LIN {X -144.015,Y -42.862,Z -106.683,A -90.000,B 90.000,C 0.000} C_DIS
LIN {X -41.460,Y -42.862,Z -106.683,A -90.000,B 90.000,C 0.000} C_DIS
LIN {X -41.247,Y -42.862,Z -104.786,A -90.000,B 90.000,C 0.000} C_DIS
LIN {X -40.987,Y -42.862,Z -102.895,A -90.000,B 90.000,C 0.000} C_DIS
LIN {X -40.681,Y -42.862,Z -101.010,A -90.000,B 90.000,C 0.000} C_DIS
LIN {X -40.328,Y -42.862,Z -99.134,A -90.000,B 90.000,C 0.000} C_DIS
LIN {X -144.015,Y -42.862,Z -99.134,A -90.000,B 90.000,C 0.000} C_DIS
LIN {X -144.015,Y -42.862,Z -91.586,A -90.000,B 90.000,C 0.000} C_DIS
LIN {X -38.308,Y -42.862,Z -91.586,A -90.000,B 90.000,C 0.000} C_DIS
LIN {X -37.692,Y -42.862,Z -90.026,A -90.000,B 90.000,C 0.000} C_DIS
LIN {X -37.020,Y -42.862,Z -88.489,A -90.000,B 90.000,C 0.000} C_DIS
LIN {X -36.293,Y -42.862,Z -86.977,A -90.000,B 90.000,C 0.000} C_DIS
LIN {X -35.511,Y -42.862,Z -85.492,A -90.000,B 90.000,C 0.000} C_DIS
LIN {X -34.677,Y -42.862,Z -84.037,A -90.000,B 90.000,C 0.000} C_DIS
LIN {X -144.015,Y -42.862,Z -84.037,A -90.000,B 90.000,C 0.000} C_DIS
LIN {X -144.015,Y -42.862,Z -76.488,A -90.000,B 90.000,C 0.000} C_DIS
LIN {X -29.075,Y -42.862,Z -76.488,A -90.000,B 90.000,C 0.000} C_DIS
LIN {X -28.227,Y -42.862,Z -75.567,A -90.000,B 90.000,C 0.000} C_DIS
LIN {X -27.332,Y -42.862,Z -74.692,A -90.000,B 90.000,C 0.000} C_DIS
LIN {X -26.392,Y -42.862,Z -73.865,A -90.000,B 90.000,C 0.000} C_DIS
LIN {X -25.410,Y -42.862,Z -73.089,A -90.000,B 90.000,C 0.000} C_DIS
LIN {X -24.388,Y -42.862,Z -72.366,A -90.000,B 90.000,C 0.000} C_DIS
LIN {X -23.329,Y -42.862,Z -71.698,A -90.000,B 90.000,C 0.000} C_DIS
LIN {X -22.236,Y -42.862,Z -71.087,A -90.000,B 90.000,C 0.000} C_DIS
LIN {X -21.113,Y -42.862,Z -70.535,A -90.000,B 90.000,C 0.000} C_DIS
LIN {X -19.962,Y -42.862,Z -70.043,A -90.000,B 90.000,C 0.000} C_DIS
LIN {X -18.787,Y -42.862,Z -69.612,A -90.000,B 90.000,C 0.000} C_DIS
LIN {X -17.590,Y -42.862,Z -69.244,A -90.000,B 90.000,C 0.000} C_DIS
LIN {X -16.376,Y -42.862,Z -68.939,A -90.000,B 90.000,C 0.000} C_DIS
LIN {X -144.015,Y -42.862,Z -68.939,A -90.000,B 90.000,C 0.000} C_DIS
LIN {X -144.015,Y -42.862,Z -61.390,A -90.000,B 90.000,C 0.000} C_DIS
LIN {X 20.649,Y -42.862,Z -61.390,A -90.000,B 90.000,C 0.000} C_DIS
LIN {X 20.813,Y -42.862,Z -60.536,A -90.000,B 90.000,C 0.000} C_DIS
LIN {X 21.035,Y -42.862,Z -59.695,A -90.000,B 90.000,C 0.000} C_DIS
LIN {X 21.313,Y -42.862,Z -58.871,A -90.000,B 90.000,C 0.000} C_DIS
LIN {X 21.646,Y -42.862,Z -58.068,A -90.000,B 90.000,C 0.000} C_DIS
LIN {X 22.032,Y -42.862,Z -57.289,A -90.000,B 90.000,C 0.000} C_DIS
LIN {X 22.470,Y -42.862,Z -56.537,A -90.000,B 90.000,C 0.000} C_DIS
LIN {X 22.958,Y -42.862,Z -55.817,A -90.000,B 90.000,C 0.000} C_DIS
LIN {X 23.493,Y -42.862,Z -55.132,A -90.000,B 90.000,C 0.000} C_DIS
LIN {X 24.073,Y -42.862,Z -54.484,A -90.000,B 90.000,C 0.000} C_DIS
LIN {X 24.696,Y -42.862,Z -53.877,A -90.000,B 90.000,C 0.000} C_DIS
LIN {X 24.707,Y -42.862,Z -53.842,A -90.000,B 90.000,C 0.000} C_DIS
LIN {X -144.015,Y -42.862,Z -53.842,A -90.000,B 90.000,C 0.000} C_DIS
LIN {X -144.015,Y -42.862,Z -46.293,A -90.000,B 90.000,C 0.000} C_DIS
LIN {X 29.758,Y -42.862,Z -46.293,A -90.000,B 90.000,C 0.000} C_DIS
LIN {X 30.551,Y -42.862,Z -45.689,A -90.000,B 90.000,C 0.000} C_DIS
LIN {X 31.381,Y -42.862,Z -45.138,A -90.000,B 90.000,C 0.000} C_DIS
LIN {X 32.246,Y -42.862,Z -44.643,A -90.000,B 90.000,C 0.000} C_DIS
LIN {X 33.142,Y -42.862,Z -44.206,A -90.000,B 90.000,C 0.000} C_DIS
LIN {X 34.064,Y -42.862,Z -43.828,A -90.000,B 90.000,C 0.000} C_DIS
LIN {X 35.010,Y -42.862,Z -43.513,A -90.000,B 90.000,C 0.000} C_DIS
LIN {X 35.974,Y -42.862,Z -43.260,A -90.000,B 90.000,C 0.000} C_DIS
LIN {X 37.013,Y -42.862,Z -43.088,A -90.000,B 90.000,C 0.000} C_DIS
LIN {X 38.061,Y -42.862,Z -42.978,A -90.000,B 90.000,C 0.000} C_DIS
LIN {X 39.113,Y -42.862,Z -42.931,A -90.000,B 90.000,C 0.000} C_DIS
LIN {X 40.166,Y -42.862,Z -42.946,A -90.000,B 90.000,C 0.000} C_DIS
LIN {X 41.217,Y -42.862,Z -43.023,A -90.000,B 90.000,C 0.000} C_DIS
LIN {X 42.261,Y -42.862,Z -43.163,A -90.000,B 90.000,C 0.000} C_DIS
LIN {X 43.295,Y -42.862,Z -43.364,A -90.000,B 90.000,C 0.000} C_DIS
LIN {X 44.315,Y -42.862,Z -43.626,A -90.000,B 90.000,C 0.000} C_DIS
LIN {X 45.317,Y -42.862,Z -43.948,A -90.000,B 90.000,C 0.000} C_DIS
LIN {X 46.299,Y -42.862,Z -44.329,A -90.000,B 90.000,C 0.000} C_DIS
LIN {X 47.257,Y -42.862,Z -44.768,A -90.000,B 90.000,C 0.000} C_DIS
LIN {X 48.087,Y -42.862,Z -44.686,A -90.000,B 90.000,C 0.000} C_DIS
LIN {X 48.921,Y -42.862,Z -44.656,A -90.000,B 90.000,C 0.000} C_DIS
LIN {X 49.755,Y -42.862,Z -44.677,A -90.000,B 90.000,C 0.000} C_DIS
LIN {X 50.586,Y -42.862,Z -44.750,A -90.000,B 90.000,C 0.000} C_DIS
LIN {X 51.357,Y -42.862,Z -44.828,A -90.000,B 90.000,C 0.000} C_DIS
LIN {X 52.122,Y -42.862,Z -44.958,A -90.000,B 90.000,C 0.000} C_DIS
LIN {X 52.876,Y -42.862,Z -45.137,A -90.000,B 90.000,C 0.000} C_DIS
LIN {X 53.616,Y -42.862,Z -45.367,A -90.000,B 90.000,C 0.000} C_DIS
LIN {X 54.330,Y -42.862,Z -45.538,A -90.000,B 90.000,C 0.000} C_DIS
LIN {X 55.034,Y -42.862,Z -45.750,A -90.000,B 90.000,C 0.000} C_DIS
LIN {X 55.724,Y -42.862,Z -46.002,A -90.000,B 90.000,C 0.000} C_DIS
LIN {X 56.398,Y -42.862,Z -46.293,A -90.000,B 90.000,C 0.000} C_DIS
LIN {X 86.662,Y -42.862,Z -46.293,A -90.000,B 90.000,C 0.000} C_DIS
LIN {X 85.043,Y -42.862,Z -47.710,A -90.000,B 90.000,C 0.000} C_DIS
LIN {X 83.466,Y -42.862,Z -49.175,A -90.000,B 90.000,C 0.000} C_DIS
LIN {X 81.935,Y -42.862,Z -50.686,A -90.000,B 90.000,C 0.000} C_DIS
LIN {X 80.449,Y -42.862,Z -52.242,A -90.000,B 90.000,C 0.000} C_DIS
LIN {X 79.010,Y -42.862,Z -53.842,A -90.000,B 90.000,C 0.000} C_DIS
LIN {X 64.970,Y -42.862,Z -53.842,A -90.000,B 90.000,C 0.000} C_DIS
LIN {X 65.683,Y -42.862,Z -54.842,A -90.000,B 90.000,C 0.000} C_DIS
LIN {X 66.353,Y -42.862,Z -55.871,A -90.000,B 90.000,C 0.000} C_DIS
LIN {X 66.978,Y -42.862,Z -56.928,A -90.000,B 90.000,C 0.000} C_DIS
LIN {X 67.558,Y -42.862,Z -58.010,A -90.000,B 90.000,C 0.000} C_DIS
LIN {X 68.092,Y -42.862,Z -59.116,A -90.000,B 90.000,C 0.000} C_DIS
LIN {X 68.578,Y -42.862,Z -60.243,A -90.000,B 90.000,C 0.000} C_DIS
LIN {X 69.017,Y -42.862,Z -61.390,A -90.000,B 90.000,C 0.000} C_DIS
LIN {X 73.958,Y -42.862,Z -61.390,A -90.000,B 90.000,C 0.000} C_DIS
LIN {X 74.651,Y -42.862,Z -60.082,A -90.000,B 90.000,C 0.000} C_DIS
LIN {X 75.393,Y -42.862,Z -58.802,A -90.000,B 90.000,C 0.000} C_DIS
LIN {X 76.183,Y -42.862,Z -57.550,A -90.000,B 90.000,C 0.000} C_DIS
LIN {X 77.020,Y -42.862,Z -56.330,A -90.000,B 90.000,C 0.000} C_DIS
LIN {X 77.903,Y -42.862,Z -55.142,A -90.000,B 90.000,C 0.000} C_DIS
LIN {X 79.161,Y -42.862,Z -53.670,A -90.000,B 90.000,C 0.000} C_DIS
LIN {X 80.458,Y -42.862,Z -52.232,A -90.000,B 90.000,C 0.000} C_DIS
LIN {X 81.794,Y -42.862,Z -50.830,A -90.000,B 90.000,C 0.000} C_DIS
LIN {X 83.166,Y -42.862,Z -49.464,A -90.000,B 90.000,C 0.000} C_DIS
LIN {X 84.575,Y -42.862,Z -48.136,A -90.000,B 90.000,C 0.000} C_DIS
LIN {X 86.019,Y -42.862,Z -46.846,A -90.000,B 90.000,C 0.000} C_DIS
LIN {X 87.497,Y -42.862,Z -45.595,A -90.000,B 90.000,C 0.000} C_DIS
LIN {X 88.554,Y -42.862,Z -44.745,A -90.000,B 90.000,C 0.000} C_DIS
LIN {X 89.585,Y -42.862,Z -43.865,A -90.000,B 90.000,C 0.000} C_DIS
LIN {X 90.592,Y -42.862,Z -42.956,A -90.000,B 90.000,C 0.000} C_DIS
LIN {X 91.572,Y -42.862,Z -42.019,A -90.000,B 90.000,C 0.000} C_DIS
LIN {X 94.550,Y -42.862,Z -38.744,A -90.000,B 90.000,C 0.000} C_DIS
LIN {X -144.015,Y -42.862,Z -38.744,A -90.000,B 90.000,C 0.000} C_DIS
LIN {X -144.015,Y -42.862,Z -31.195,A -90.000,B 90.000,C 0.000} C_DIS
LIN {X 102.214,Y -42.862,Z -31.195,A -90.000,B 90.000,C 0.000} C_DIS
LIN {X 103.051,Y -42.862,Z -30.607,A -90.000,B 90.000,C 0.000} C_DIS
LIN {X 103.927,Y -42.862,Z -30.078,A -90.000,B 90.000,C 0.000} C_DIS
LIN {X 104.837,Y -42.862,Z -29.611,A -90.000,B 90.000,C 0.000} C_DIS
LIN {X 105.777,Y -42.862,Z -29.208,A -90.000,B 90.000,C 0.000} C_DIS
LIN {X 106.743,Y -42.862,Z -28.871,A -90.000,B 90.000,C 0.000} C_DIS
LIN {X 107.730,Y -42.862,Z -28.602,A -90.000,B 90.000,C 0.000} C_DIS
LIN {X 108.733,Y -42.862,Z -28.401,A -90.000,B 90.000,C 0.000} C_DIS
LIN {X 109.747,Y -42.862,Z -28.270,A -90.000,B 90.000,C 0.000} C_DIS
LIN {X 110.768,Y -42.862,Z -28.209,A -90.000,B 90.000,C 0.000} C_DIS
LIN {X 111.791,Y -42.862,Z -28.219,A -90.000,B 90.000,C 0.000} C_DIS
LIN {X 112.811,Y -42.862,Z -28.301,A -90.000,B 90.000,C 0.000} C_DIS
LIN {X 112.936,Y -42.862,Z -28.324,A -90.000,B 90.000,C 0.000} C_DIS
LIN {X 112.988,Y -42.862,Z -28.327,A -90.000,B 90.000,C 0.000} C_DIS
LIN {X 113.926,Y -42.862,Z -28.470,A -90.000,B 90.000,C 0.000} C_DIS
LIN {X 114.851,Y -42.862,Z -28.677,A -90.000,B 90.000,C 0.000} C_DIS
LIN {X 115.760,Y -42.862,Z -28.948,A -90.000,B 90.000,C 0.000} C_DIS
LIN {X 116.648,Y -42.862,Z -29.280,A -90.000,B 90.000,C 0.000} C_DIS
LIN {X 117.511,Y -42.862,Z -29.673,A -90.000,B 90.000,C 0.000} C_DIS
LIN {X 118.345,Y -42.862,Z -30.125,A -90.000,B 90.000,C 0.000} C_DIS
LIN {X 119.146,Y -42.862,Z -30.633,A -90.000,B 90.000,C 0.000} C_DIS
LIN {X 119.910,Y -42.862,Z -31.195,A -90.000,B 90.000,C 0.000} C_DIS
LIN {X 144.015,Y -42.862,Z -31.195,A -90.000,B 90.000,C 0.000} C_DIS
LIN {X 144.015,Y -42.862,Z -38.744,A -90.000,B 90.000,C 0.000} C_DIS
LIN {X 124.744,Y -42.862,Z -38.744,A -90.000,B 90.000,C 0.000} C_DIS
LIN {X 124.926,Y -42.862,Z -39.587,A -90.000,B 90.000,C 0.000} C_DIS
LIN {X 125.057,Y -42.862,Z -40.439,A -90.000,B 90.000,C 0.000} C_DIS
LIN {X 125.135,Y -42.862,Z -41.298,A -90.000,B 90.000,C 0.000} C_DIS
LIN {X 125.160,Y -42.862,Z -42.159,A -90.000,B 90.000,C 0.000} C_DIS
LIN {X 125.132,Y -42.862,Z -43.021,A -90.000,B 90.000,C 0.000} C_DIS
LIN {X 124.953,Y -42.862,Z -44.119,A -90.000,B 90.000,C 0.000} C_DIS
LIN {X 124.737,Y -42.862,Z -45.210,A -90.000,B 90.000,C 0.000} C_DIS
LIN {X 124.482,Y -42.862,Z -46.293,A -90.000,B 90.000,C 0.000} C_DIS
LIN {X 144.015,Y -42.862,Z -46.293,A -90.000,B 90.000,C 0.000} C_DIS
LIN {X 144.015,Y -42.862,Z -53.842,A -90.000,B 90.000,C 0.000} C_DIS
LIN {X 121.443,Y -42.862,Z -53.842,A -90.000,B 90.000,C 0.000} C_DIS
LIN {X 120.742,Y -42.862,Z -55.297,A -90.000,B 90.000,C 0.000} C_DIS
LIN {X 120.079,Y -42.862,Z -56.770,A -90.000,B 90.000,C 0.000} C_DIS
LIN {X 119.457,Y -42.862,Z -58.260,A -90.000,B 90.000,C 0.000} C_DIS
LIN {X 118.875,Y -42.862,Z -59.766,A -90.000,B 90.000,C 0.000} C_DIS
LIN {X 118.368,Y -42.862,Z -61.390,A -90.000,B 90.000,C 0.000} C_DIS
LIN {X 144.015,Y -42.862,Z -61.390,A -90.000,B 90.000,C 0.000} C_DIS
LIN {X 144.015,Y -42.862,Z -68.939,A -90.000,B 90.000,C 0.000} C_DIS
LIN {X 115.738,Y -42.862,Z -68.939,A -90.000,B 90.000,C 0.000} C_DIS
LIN {X 115.018,Y -42.862,Z -70.802,A -90.000,B 90.000,C 0.000} C_DIS
LIN {X 114.272,Y -42.862,Z -72.655,A -90.000,B 90.000,C 0.000} C_DIS
LIN {X 113.767,Y -42.862,Z -73.946,A -90.000,B 90.000,C 0.000} C_DIS
LIN {X 113.230,Y -42.862,Z -75.224,A -90.000,B 90.000,C 0.000} C_DIS
LIN {X 112.660,Y -42.862,Z -76.488,A -90.000,B 90.000,C 0.000} C_DIS
LIN {X 144.015,Y -42.862,Z -76.488,A -90.000,B 90.000,C 0.000} C_DIS
LIN {X 144.015,Y -42.862,Z -84.037,A -90.000,B 90.000,C 0.000} C_DIS
LIN {X 108.391,Y -42.862,Z -84.037,A -90.000,B 90.000,C 0.000} C_DIS
LIN {X 107.637,Y -42.862,Z -85.126,A -90.000,B 90.000,C 0.000} C_DIS
LIN {X 106.857,Y -42.862,Z -86.197,A -90.000,B 90.000,C 0.000} C_DIS
LIN {X 106.156,Y -42.862,Z -87.168,A -90.000,B 90.000,C 0.000} C_DIS
LIN {X 105.419,Y -42.862,Z -88.112,A -90.000,B 90.000,C 0.000} C_DIS
LIN {X 104.647,Y -42.862,Z -89.027,A -90.000,B 90.000,C 0.000} C_DIS
LIN {X 103.840,Y -42.862,Z -89.911,A -90.000,B 90.000,C 0.000} C_DIS
LIN {X 103.001,Y -42.862,Z -90.765,A -90.000,B 90.000,C 0.000} C_DIS
LIN {X 102.129,Y -42.862,Z -91.586,A -90.000,B 90.000,C 0.000} C_DIS
LIN {X 144.015,Y -42.862,Z -91.586,A -90.000,B 90.000,C 0.000} C_DIS
LIN {X 144.015,Y -42.862,Z -99.134,A -90.000,B 90.000,C 0.000} C_DIS
LIN {X 99.151,Y -42.862,Z -99.134,A -90.000,B 90.000,C 0.000} C_DIS
LIN {X 98.860,Y -42.862,Z -100.099,A -90.000,B 90.000,C 0.000} C_DIS
LIN {X 98.506,Y -42.862,Z -101.043,A -90.000,B 90.000,C 0.000} C_DIS
LIN {X 98.089,Y -42.862,Z -101.961,A -90.000,B 90.000,C 0.000} C_DIS
LIN {X 97.612,Y -42.862,Z -102.849,A -90.000,B 90.000,C 0.000} C_DIS
LIN {X 97.077,Y -42.862,Z -103.703,A -90.000,B 90.000,C 0.000} C_DIS
LIN {X 96.485,Y -42.862,Z -104.519,A -90.000,B 90.000,C 0.000} C_DIS
LIN {X 95.841,Y -42.862,Z -105.294,A -90.000,B 90.000,C 0.000} C_DIS
LIN {X 95.901,Y -42.862,Z -105.988,A -90.000,B 90.000,C 0.000} C_DIS
LIN {X 95.943,Y -42.862,Z -106.683,A -90.000,B 90.000,C 0.000} C_DIS
LIN {X 144.015,Y -42.862,Z -106.683,A -90.000,B 90.000,C 0.000} C_DIS
LIN {X 144.015,Y -42.862,Z -114.232,A -90.000,B 90.000,C 0.000} C_DIS
LIN {X 95.004,Y -42.862,Z -114.232,A -90.000,B 90.000,C 0.000} C_DIS
LIN {X 94.755,Y -42.862,Z -115.216,A -90.000,B 90.000,C 0.000} C_DIS
LIN {X 94.481,Y -42.862,Z -116.194,A -90.000,B 90.000,C 0.000} C_DIS
LIN {X 94.133,Y -42.862,Z -117.126,A -90.000,B 90.000,C 0.000} C_DIS
LIN {X 93.819,Y -42.862,Z -118.070,A -90.000,B 90.000,C 0.000} C_DIS
LIN {X 93.540,Y -42.862,Z -119.025,A -90.000,B 90.000,C 0.000} C_DIS
LIN {X 93.683,Y -42.862,Z -119.949,A -90.000,B 90.000,C 0.000} C_DIS
LIN {X 93.853,Y -42.862,Z -120.868,A -90.000,B 90.000,C 0.000} C_DIS
LIN {X 94.052,Y -42.862,Z -121.781,A -90.000,B 90.000,C 0.000} C_DIS
LIN {X 144.015,Y -42.862,Z -121.781,A -90.000,B 90.000,C 0.000} C_DIS
LIN {X 144.015,Y -42.862,Z -129.329,A -90.000,B 90.000,C 0.000} C_DIS
LIN {X 94.517,Y -42.862,Z -129.329,A -90.000,B 90.000,C 0.000} C_DIS
LIN {X 94.482,Y -42.862,Z -130.307,A -90.000,B 90.000,C 0.000} C_DIS
LIN {X 94.426,Y -42.862,Z -131.284,A -90.000,B 90.000,C 0.000} C_DIS
LIN {X 94.348,Y -42.862,Z -132.259,A -90.000,B 90.000,C 0.000} C_DIS
LIN {X 94.250,Y -42.862,Z -134.569,A -90.000,B 90.000,C 0.000} C_DIS
LIN {X 94.147,Y -42.862,Z -136.878,A -90.000,B 90.000,C 0.000} C_DIS
LIN {X 144.015,Y -42.862,Z -136.878,A -90.000,B 90.000,C 0.000} C_DIS
LIN {X 144.015,Y -42.862,Z -144.427,A -90.000,B 90.000,C 0.000} C_DIS
LIN {X 93.773,Y -42.862,Z -144.427,A -90.000,B 90.000,C 0.000} C_DIS
LIN {X 93.759,Y -42.862,Z -144.687,A -90.000,B 90.000,C 0.000} C_DIS
LIN {X 93.660,Y -42.862,Z -146.513,A -90.000,B 90.000,C 0.000} C_DIS
LIN {X 93.529,Y -42.862,Z -148.337,A -90.000,B 90.000,C 0.000} C_DIS
LIN {X 93.366,Y -42.862,Z -150.158,A -90.000,B 90.000,C 0.000} C_DIS
LIN {X 93.171,Y -42.862,Z -151.976,A -90.000,B 90.000,C 0.000} C_DIS
LIN {X 144.015,Y -42.862,Z -151.976,A -90.000,B 90.000,C 0.000} C_DIS
LIN {X 144.015,Y -42.862,Z -159.525,A -90.000,B 90.000,C 0.000} C_DIS
LIN {X 92.013,Y -42.862,Z -159.525,A -90.000,B 90.000,C 0.000} C_DIS
LIN {X 91.632,Y -42.862,Z -161.424,A -90.000,B 90.000,C 0.000} C_DIS
LIN {X 91.216,Y -42.862,Z -163.315,A -90.000,B 90.000,C 0.000} C_DIS
LIN {X 90.765,Y -42.862,Z -165.198,A -90.000,B 90.000,C 0.000} C_DIS
LIN {X 90.279,Y -42.862,Z -167.073,A -90.000,B 90.000,C 0.000} C_DIS
LIN {X 144.015,Y -42.862,Z -167.073,A -90.000,B 90.000,C 0.000} C_DIS
LIN {X 144.015,Y -42.862,Z -174.622,A -90.000,B 90.000,C 0.000} C_DIS
LIN {X 87.981,Y -42.862,Z -174.622,A -90.000,B 90.000,C 0.000} C_DIS
LIN {X 87.289,Y -42.862,Z -176.815,A -90.000,B 90.000,C 0.000} C_DIS
LIN {X 86.606,Y -42.862,Z -179.011,A -90.000,B 90.000,C 0.000} C_DIS
LIN {X 85.836,Y -42.862,Z -182.171,A -90.000,B 90.000,C 0.000} C_DIS
LIN {X 144.015,Y -42.862,Z -182.171,A -90.000,B 90.000,C 0.000} C_DIS
LIN {X 144.015,Y -42.862,Z -189.720,A -90.000,B 90.000,C 0.000} C_DIS
LIN {X 83.918,Y -42.862,Z -189.720,A -90.000,B 90.000,C 0.000} C_DIS
LIN {X 83.235,Y -42.862,Z -192.307,A -90.000,B 90.000,C 0.000} C_DIS
LIN {X 82.539,Y -42.862,Z -194.890,A -90.000,B 90.000,C 0.000} C_DIS
LIN {X 82.150,Y -42.862,Z -196.080,A -90.000,B 90.000,C 0.000} C_DIS
LIN {X 81.756,Y -42.862,Z -197.269,A -90.000,B 90.000,C 0.000} C_DIS
LIN {X 144.015,Y -42.862,Z -197.269,A -90.000,B 90.000,C 0.000} C_DIS
LIN {X 144.015,Y -42.862,Z -204.817,A -90.000,B 90.000,C 0.000} C_DIS
LIN {X 79.114,Y -42.862,Z -204.817,A -90.000,B 90.000,C 0.000} C_DIS
LIN {X 78.176,Y -42.862,Z -207.342,A -90.000,B 90.000,C 0.000} C_DIS
LIN {X 77.215,Y -42.862,Z -209.859,A -90.000,B 90.000,C 0.000} C_DIS
LIN {X 76.229,Y -42.862,Z -212.366,A -90.000,B 90.000,C 0.000} C_DIS
LIN {X 144.015,Y -42.862,Z -212.366,A -90.000,B 90.000,C 0.000} C_DIS
LIN {X 144.015,Y -42.862,Z -219.915,A -90.000,B 90.000,C 0.000} C_DIS
LIN {X 73.092,Y -42.862,Z -219.915,A -90.000,B 90.000,C 0.000} C_DIS
LIN {X 71.984,Y -42.862,Z -222.442,A -90.000,B 90.000,C 0.000} C_DIS
LIN {X 70.851,Y -42.862,Z -224.959,A -90.000,B 90.000,C 0.000} C_DIS
LIN {X 69.694,Y -42.862,Z -227.464,A -90.000,B 90.000,C 0.000} C_DIS
LIN {X 144.015,Y -42.862,Z -227.464,A -90.000,B 90.000,C 0.000} C_DIS
LIN {X 144.015,Y -42.862,Z -235.012,A -90.000,B 90.000,C 0.000} C_DIS
LIN {X 66.063,Y -42.862,Z -235.012,A -90.000,B 90.000,C 0.000} C_DIS
LIN {X 65.077,Y -42.862,Z -236.924,A -90.000,B 90.000,C 0.000} C_DIS
LIN {X 64.061,Y -42.862,Z -238.820,A -90.000,B 90.000,C 0.000} C_DIS
LIN {X 63.015,Y -42.862,Z -240.699,A -90.000,B 90.000,C 0.000} C_DIS
LIN {X 61.939,Y -42.862,Z -242.561,A -90.000,B 90.000,C 0.000} C_DIS
LIN {X 144.015,Y -42.862,Z -242.561,A -90.000,B 90.000,C 0.000} C_DIS
LIN {X 144.015,Y -42.862,Z -23.646,A -90.000,B 90.000,C 0.000} C_DIS
LIN {X -144.015,Y -42.862,Z -23.646,A -90.000,B 90.000,C 0.000} C_DIS
LIN {X -144.015,Y -42.862,Z -16.098,A -90.000,B 90.000,C 0.000} C_DIS
LIN {X 144.015,Y -42.862,Z -16.098,A -90.000,B 90.000,C 0.000} C_DIS
LIN {X 144.015,Y -42.862,Z -8.549,A -90.000,B 90.000,C 0.000} C_DIS
LIN {X -144.015,Y -42.862,Z -8.549,A -90.000,B 90.000,C 0.000} C_DIS
LIN {X -144.015,Y -42.862,Z -1.000,A -90.000,B 90.000,C 0.000} C_DIS
LIN {X 144.015,Y -42.862,Z -1.000,A -90.000,B 90.000,C 0.000} C_DIS
LIN {X 55.699,Y -42.862,Z -45.992,A -90.000,B 90.000,C 0.000} C_DIS
LIN {X 55.017,Y -42.862,Z -45.744,A -90.000,B 90.000,C 0.000} C_DIS
LIN {X 54.322,Y -42.862,Z -45.536,A -90.000,B 90.000,C 0.000} C_DIS
LIN {X 53.616,Y -42.862,Z -45.367,A -90.000,B 90.000,C 0.000} C_DIS
LIN {X 52.876,Y -42.862,Z -45.138,A -90.000,B 90.000,C 0.000} C_DIS
LIN {X 52.121,Y -42.862,Z -44.958,A -90.000,B 90.000,C 0.000} C_DIS
LIN {X 51.357,Y -42.862,Z -44.829,A -90.000,B 90.000,C 0.000} C_DIS
LIN {X 50.586,Y -42.862,Z -44.750,A -90.000,B 90.000,C 0.000} C_DIS
LIN {X 49.755,Y -42.862,Z -44.677,A -90.000,B 90.000,C 0.000} C_DIS
LIN {X 48.921,Y -42.862,Z -44.656,A -90.000,B 90.000,C 0.000} C_DIS
LIN {X 48.087,Y -42.862,Z -44.687,A -90.000,B 90.000,C 0.000} C_DIS
LIN {X 47.257,Y -42.862,Z -44.768,A -90.000,B 90.000,C 0.000} C_DIS
LIN {X 46.299,Y -42.862,Z -44.329,A -90.000,B 90.000,C 0.000} C_DIS
LIN {X 45.317,Y -42.862,Z -43.948,A -90.000,B 90.000,C 0.000} C_DIS
LIN {X 44.315,Y -42.862,Z -43.626,A -90.000,B 90.000,C 0.000} C_DIS
LIN {X 43.295,Y -42.862,Z -43.364,A -90.000,B 90.000,C 0.000} C_DIS
LIN {X 42.261,Y -42.862,Z -43.163,A -90.000,B 90.000,C 0.000} C_DIS
LIN {X 41.217,Y -42.862,Z -43.023,A -90.000,B 90.000,C 0.000} C_DIS
LIN {X 40.166,Y -42.862,Z -42.946,A -90.000,B 90.000,C 0.000} C_DIS
LIN {X 39.113,Y -42.862,Z -42.931,A -90.000,B 90.000,C 0.000} C_DIS
LIN {X 38.061,Y -42.862,Z -42.978,A -90.000,B 90.000,C 0.000} C_DIS
LIN {X 37.013,Y -42.862,Z -43.088,A -90.000,B 90.000,C 0.000} C_DIS
LIN {X 35.974,Y -42.862,Z -43.260,A -90.000,B 90.000,C 0.000} C_DIS
LIN {X 34.989,Y -42.862,Z -43.519,A -90.000,B 90.000,C 0.000} C_DIS
LIN {X 34.023,Y -42.862,Z -43.844,A -90.000,B 90.000,C 0.000} C_DIS
LIN {X 33.082,Y -42.862,Z -44.233,A -90.000,B 90.000,C 0.000} C_DIS
LIN {X 32.168,Y -42.862,Z -44.684,A -90.000,B 90.000,C 0.000} C_DIS
LIN {X 31.287,Y -42.862,Z -45.196,A -90.000,B 90.000,C 0.000} C_DIS
LIN {X 30.443,Y -42.862,Z -45.766,A -90.000,B 90.000,C 0.000} C_DIS
LIN {X 29.639,Y -42.862,Z -46.391,A -90.000,B 90.000,C 0.000} C_DIS
LIN {X 28.879,Y -42.862,Z -47.069,A -90.000,B 90.000,C 0.000} C_DIS
LIN {X 28.166,Y -42.862,Z -47.797,A -90.000,B 90.000,C 0.000} C_DIS
LIN {X 27.503,Y -42.862,Z -48.571,A -90.000,B 90.000,C 0.000} C_DIS
LIN {X 26.894,Y -42.862,Z -49.388,A -90.000,B 90.000,C 0.000} C_DIS
LIN {X 26.342,Y -42.862,Z -50.244,A -90.000,B 90.000,C 0.000} C_DIS
LIN {X 25.848,Y -42.862,Z -51.135,A -90.000,B 90.000,C 0.000} C_DIS
LIN {X 25.415,Y -42.862,Z -52.057,A -90.000,B 90.000,C 0.000} C_DIS
LIN {X 25.138,Y -42.862,Z -52.649,A -90.000,B 90.000,C 0.000} C_DIS
LIN {X 24.898,Y -42.862,Z -53.256,A -90.000,B 90.000,C 0.000} C_DIS
LIN {X 24.696,Y -42.862,Z -53.877,A -90.000,B 90.000,C 0.000} C_DIS
LIN {X 24.058,Y -42.862,Z -54.500,A -90.000,B 90.000,C 0.000} C_DIS
LIN {X 23.464,Y -42.862,Z -55.167,A -90.000,B 90.000,C 0.000} C_DIS
LIN {X 22.918,Y -42.862,Z -55.872,A -90.000,B 90.000,C 0.000} C_DIS
LIN {X 22.422,Y -42.862,Z -56.614,A -90.000,B 90.000,C 0.000} C_DIS
LIN {X 21.979,Y -42.862,Z -57.388,A -90.000,B 90.000,C 0.000} C_DIS
LIN {X 21.590,Y -42.862,Z -58.191,A -90.000,B 90.000,C 0.000} C_DIS
LIN {X 21.258,Y -42.862,Z -59.020,A -90.000,B 90.000,C 0.000} C_DIS
LIN {X 20.984,Y -42.862,Z -59.869,A -90.000,B 90.000,C 0.000} C_DIS
LIN {X 20.770,Y -42.862,Z -60.735,A -90.000,B 90.000,C 0.000} C_DIS
LIN {X 20.616,Y -42.862,Z -61.614,A -90.000,B 90.000,C 0.000} C_DIS
LIN {X 20.523,Y -42.862,Z -62.501,A -90.000,B 90.000,C 0.000} C_DIS
LIN {X 19.836,Y -42.862,Z -62.571,A -90.000,B 90.000,C 0.000} C_DIS
LIN {X 19.155,Y -42.862,Z -62.686,A -90.000,B 90.000,C 0.000} C_DIS
LIN {X 18.482,Y -42.862,Z -62.843,A -90.000,B 90.000,C 0.000} C_DIS
LIN {X 18.425,Y -42.862,Z -62.863,A -90.000,B 90.000,C 0.000} C_DIS
LIN {X 17.595,Y -42.862,Z -63.039,A -90.000,B 90.000,C 0.000} C_DIS
LIN {X 16.783,Y -42.862,Z -63.284,A -90.000,B 90.000,C 0.000} C_DIS
LIN {X 15.994,Y -42.862,Z -63.595,A -90.000,B 90.000,C 0.000} C_DIS
LIN {X 15.234,Y -42.862,Z -63.970,A -90.000,B 90.000,C 0.000} C_DIS
LIN {X 14.507,Y -42.862,Z -64.408,A -90.000,B 90.000,C 0.000} C_DIS
LIN {X 13.820,Y -42.862,Z -64.904,A -90.000,B 90.000,C 0.000} C_DIS
LIN {X 13.176,Y -42.862,Z -65.456,A -90.000,B 90.000,C 0.000} C_DIS
LIN {X 12.579,Y -42.862,Z -66.059,A -90.000,B 90.000,C 0.000} C_DIS
LIN {X 12.036,Y -42.862,Z -66.710,A -90.000,B 90.000,C 0.000} C_DIS
LIN {X 11.548,Y -42.862,Z -67.404,A -90.000,B 90.000,C 0.000} C_DIS
LIN {X 11.223,Y -42.862,Z -67.900,A -90.000,B 90.000,C 0.000} C_DIS
LIN {X 10.925,Y -42.862,Z -68.412,A -90.000,B 90.000,C 0.000} C_DIS
LIN {X 10.655,Y -42.862,Z -68.939,A -90.000,B 90.000,C 0.000} C_DIS
LIN {X -4.102,Y -42.862,Z -68.939,A -90.000,B 90.000,C 0.000} C_DIS
LIN {X -7.573,Y -42.862,Z -69.409,A -90.000,B 90.000,C 0.000} C_DIS
LIN {X -4.519,Y -42.862,Z -69.884,A -90.000,B 90.000,C 0.000} C_DIS
LIN {X -1.474,Y -42.862,Z -70.415,A -90.000,B 90.000,C 0.000} C_DIS
LIN {X 1.560,Y -42.862,Z -71.004,A -90.000,B 90.000,C 0.000} C_DIS
LIN {X 4.583,Y -42.862,Z -71.648,A -90.000,B 90.000,C 0.000} C_DIS
LIN {X 7.593,Y -42.862,Z -72.349,A -90.000,B 90.000,C 0.000} C_DIS
LIN {X 10.590,Y -42.862,Z -73.106,A -90.000,B 90.000,C 0.000} C_DIS
LIN {X 10.668,Y -42.862,Z -72.322,A -90.000,B 90.000,C 0.000} C_DIS
LIN {X 10.808,Y -42.862,Z -71.546,A -90.000,B 90.000,C 0.000} C_DIS
LIN {X 11.007,Y -42.862,Z -70.784,A -90.000,B 90.000,C 0.000} C_DIS
LIN {X 11.266,Y -42.862,Z -70.040,A -90.000,B 90.000,C 0.000} C_DIS
LIN {X 11.582,Y -42.862,Z -69.318,A -90.000,B 90.000,C 0.000} C_DIS
LIN {X 11.954,Y -42.862,Z -68.623,A -90.000,B 90.000,C 0.000} C_DIS
LIN {X 12.379,Y -42.862,Z -67.960,A -90.000,B 90.000,C 0.000} C_DIS
LIN {X 12.824,Y -42.862,Z -67.326,A -90.000,B 90.000,C 0.000} C_DIS
LIN {X 13.320,Y -42.862,Z -66.731,A -90.000,B 90.000,C 0.000} C_DIS
LIN {X 13.865,Y -42.862,Z -66.181,A -90.000,B 90.000,C 0.000} C_DIS
LIN {X 14.454,Y -42.862,Z -65.678,A -90.000,B 90.000,C 0.000} C_DIS
LIN {X 15.083,Y -42.862,Z -65.226,A -90.000,B 90.000,C 0.000} C_DIS
LIN {X 15.748,Y -42.862,Z -64.829,A -90.000,B 90.000,C 0.000} C_DIS
LIN {X 16.444,Y -42.862,Z -64.489,A -90.000,B 90.000,C 0.000} C_DIS
LIN {X 17.166,Y -42.862,Z -64.209,A -90.000,B 90.000,C 0.000} C_DIS
LIN {X 17.909,Y -42.862,Z -63.991,A -90.000,B 90.000,C 0.000} C_DIS
LIN {X 18.668,Y -42.862,Z -63.836,A -90.000,B 90.000,C 0.000} C_DIS
LIN {X 18.772,Y -42.862,Z -63.801,A -90.000,B 90.000,C 0.000} C_DIS
LIN {X 19.442,Y -42.862,Z -63.648,A -90.000,B 90.000,C 0.000} C_DIS
LIN {X 20.121,Y -42.862,Z -63.543,A -90.000,B 90.000,C 0.000} C_DIS
LIN {X 20.805,Y -42.862,Z -63.486,A -90.000,B 90.000,C 0.000} C_DIS
LIN {X 21.492,Y -42.862,Z -63.477,A -90.000,B 90.000,C 0.000} C_DIS
LIN {X 21.517,Y -42.862,Z -62.624,A -90.000,B 90.000,C 0.000} C_DIS
LIN {X 21.603,Y -42.862,Z -61.775,A -90.000,B 90.000,C 0.000} C_DIS
LIN {X 21.750,Y -42.862,Z -60.934,A -90.000,B 90.000,C 0.000} C_DIS
LIN {X 21.957,Y -42.862,Z -60.106,A -90.000,B 90.000,C 0.000} C_DIS
LIN {X 22.222,Y -42.862,Z -59.294,A -90.000,B 90.000,C 0.000} C_DIS
LIN {X 22.546,Y -42.862,Z -58.504,A -90.000,B 90.000,C 0.000} C_DIS
LIN {X 22.925,Y -42.862,Z -57.740,A -90.000,B 90.000,C 0.000} C_DIS
LIN {X 23.358,Y -42.862,Z -57.004,A -90.000,B 90.000,C 0.000} C_DIS
LIN {X 23.843,Y -42.862,Z -56.302,A -90.000,B 90.000,C 0.000} C_DIS
LIN {X 24.377,Y -42.862,Z -55.636,A -90.000,B 90.000,C 0.000} C_DIS
LIN {X 24.958,Y -42.862,Z -55.010,A -90.000,B 90.000,C 0.000} C_DIS
LIN {X 25.582,Y -42.862,Z -54.428,A -90.000,B 90.000,C 0.000} C_DIS
LIN {X 25.781,Y -42.862,Z -53.762,A -90.000,B 90.000,C 0.000} C_DIS
LIN {X 26.028,Y -42.862,Z -53.112,A -90.000,B 90.000,C 0.000} C_DIS
LIN {X 26.321,Y -42.862,Z -52.481,A -90.000,B 90.000,C 0.000} C_DIS
LIN {X 26.724,Y -42.862,Z -51.618,A -90.000,B 90.000,C 0.000} C_DIS
LIN {X 27.184,Y -42.862,Z -50.783,A -90.000,B 90.000,C 0.000} C_DIS
LIN {X 27.699,Y -42.862,Z -49.982,A -90.000,B 90.000,C 0.000} C_DIS
LIN {X 28.267,Y -42.862,Z -49.217,A -90.000,B 90.000,C 0.000} C_DIS
LIN {X 28.885,Y -42.862,Z -48.492,A -90.000,B 90.000,C 0.000} C_DIS
LIN {X 29.550,Y -42.862,Z -47.810,A -90.000,B 90.000,C 0.000} C_DIS
LIN {X 30.260,Y -42.862,Z -47.175,A -90.000,B 90.000,C 0.000} C_DIS
LIN {X 31.011,Y -42.862,Z -46.588,A -90.000,B 90.000,C 0.000} C_DIS
LIN {X 31.800,Y -42.862,Z -46.054,A -90.000,B 90.000,C 0.000} C_DIS
LIN {X 32.623,Y -42.862,Z -45.574,A -90.000,B 90.000,C 0.000} C_DIS
LIN {X 33.477,Y -42.862,Z -45.151,A -90.000,B 90.000,C 0.000} C_DIS
LIN {X 34.357,Y -42.862,Z -44.786,A -90.000,B 90.000,C 0.000} C_DIS
LIN {X 35.260,Y -42.862,Z -44.481,A -90.000,B 90.000,C 0.000} C_DIS
LIN {X 36.181,Y -42.862,Z -44.239,A -90.000,B 90.000,C 0.000} C_DIS
LIN {X 37.188,Y -42.862,Z -44.074,A -90.000,B 90.000,C 0.000} C_DIS
LIN {X 38.203,Y -42.862,Z -43.971,A -90.000,B 90.000,C 0.000} C_DIS
LIN {X 39.223,Y -42.862,Z -43.930,A -90.000,B 90.000,C 0.000} C_DIS
LIN {X 40.243,Y -42.862,Z -43.951,A -90.000,B 90.000,C 0.000} C_DIS
LIN {X 41.260,Y -42.862,Z -44.034,A -90.000,B 90.000,C 0.000} C_DIS
LIN {X 42.270,Y -42.862,Z -44.179,A -90.000,B 90.000,C 0.000} C_DIS
LIN {X 43.269,Y -42.862,Z -44.385,A -90.000,B 90.000,C 0.000} C_DIS
LIN {X 44.254,Y -42.862,Z -44.651,A -90.000,B 90.000,C 0.000} C_DIS
LIN {X 45.221,Y -42.862,Z -44.977,A -90.000,B 90.000,C 0.000} C_DIS
LIN {X 46.166,Y -42.862,Z -45.362,A -90.000,B 90.000,C 0.000} C_DIS
LIN {X 47.086,Y -42.862,Z -45.803,A -90.000,B 90.000,C 0.000} C_DIS
LIN {X 47.934,Y -42.862,Z -45.701,A -90.000,B 90.000,C 0.000} C_DIS
LIN {X 48.788,Y -42.862,Z -45.658,A -90.000,B 90.000,C 0.000} C_DIS
LIN {X 49.642,Y -42.862,Z -45.673,A -90.000,B 90.000,C 0.000} C_DIS
LIN {X 50.493,Y -42.862,Z -45.746,A -90.000,B 90.000,C 0.000} C_DIS
LIN {X 51.220,Y -42.862,Z -45.819,A -90.000,B 90.000,C 0.000} C_DIS
LIN {X 51.941,Y -42.862,Z -45.942,A -90.000,B 90.000,C 0.000} C_DIS
LIN {X 52.652,Y -42.862,Z -46.113,A -90.000,B 90.000,C 0.000} C_DIS
LIN {X 53.349,Y -42.862,Z -46.333,A -90.000,B 90.000,C 0.000} C_DIS
LIN {X 54.126,Y -42.862,Z -46.519,A -90.000,B 90.000,C 0.000} C_DIS
LIN {X 54.888,Y -42.862,Z -46.757,A -90.000,B 90.000,C 0.000} C_DIS
LIN {X 55.633,Y -42.862,Z -47.046,A -90.000,B 90.000,C 0.000} C_DIS
LIN {X 56.356,Y -42.862,Z -47.385,A -90.000,B 90.000,C 0.000} C_DIS
LIN {X 57.055,Y -42.862,Z -47.772,A -90.000,B 90.000,C 0.000} C_DIS
LIN {X 57.727,Y -42.862,Z -48.204,A -90.000,B 90.000,C 0.000} C_DIS
LIN {X 58.848,Y -42.862,Z -49.026,A -90.000,B 90.000,C 0.000} C_DIS
LIN {X 59.927,Y -42.862,Z -49.904,A -90.000,B 90.000,C 0.000} C_DIS
LIN {X 60.961,Y -42.862,Z -50.833,A -90.000,B 90.000,C 0.000} C_DIS
LIN {X 61.947,Y -42.862,Z -51.813,A -90.000,B 90.000,C 0.000} C_DIS
LIN {X 62.883,Y -42.862,Z -52.841,A -90.000,B 90.000,C 0.000} C_DIS
LIN {X 63.767,Y -42.862,Z -53.914,A -90.000,B 90.000,C 0.000} C_DIS
LIN {X 64.597,Y -42.862,Z -55.030,A -90.000,B 90.000,C 0.000} C_DIS
LIN {X 65.370,Y -42.862,Z -56.186,A -90.000,B 90.000,C 0.000} C_DIS
LIN {X 66.085,Y -42.862,Z -57.378,A -90.000,B 90.000,C 0.000} C_DIS
LIN {X 66.739,Y -42.862,Z -58.605,A -90.000,B 90.000,C 0.000} C_DIS
LIN {X 67.332,Y -42.862,Z -59.863,A -90.000,B 90.000,C 0.000} C_DIS
LIN {X 67.861,Y -42.862,Z -61.148,A -90.000,B 90.000,C 0.000} C_DIS
LIN {X 68.325,Y -42.862,Z -62.459,A -90.000,B 90.000,C 0.000} C_DIS
LIN {X 68.379,Y -42.862,Z -62.632,A -90.000,B 90.000,C 0.000} C_DIS
LIN {X 68.697,Y -42.862,Z -63.294,A -90.000,B 90.000,C 0.000} C_DIS
LIN {X 69.008,Y -42.862,Z -63.959,A -90.000,B 90.000,C 0.000} C_DIS
LIN {X 69.485,Y -42.862,Z -64.748,A -90.000,B 90.000,C 0.000} C_DIS
LIN {X 69.929,Y -42.862,Z -65.556,A -90.000,B 90.000,C 0.000} C_DIS
LIN {X 70.376,Y -42.862,Z -65.908,A -90.000,B 90.000,C 0.000} C_DIS
LIN {X 70.802,Y -42.862,Z -66.285,A -90.000,B 90.000,C 0.000} C_DIS
LIN {X 71.205,Y -42.862,Z -66.686,A -90.000,B 90.000,C 0.000} C_DIS
LIN {X 71.585,Y -42.862,Z -67.110,A -90.000,B 90.000,C 0.000} C_DIS
LIN {X 71.642,Y -42.862,Z -67.188,A -90.000,B 90.000,C 0.000} C_DIS
LIN {X 71.795,Y -42.862,Z -67.275,A -90.000,B 90.000,C 0.000} C_DIS
LIN {X 72.477,Y -42.862,Z -67.745,A -90.000,B 90.000,C 0.000} C_DIS
LIN {X 72.516,Y -42.862,Z -67.561,A -90.000,B 90.000,C 0.000} C_DIS
LIN {X 72.992,Y -42.862,Z -66.153,A -90.000,B 90.000,C 0.000} C_DIS
LIN {X 73.522,Y -42.862,Z -64.765,A -90.000,B 90.000,C 0.000} C_DIS
LIN {X 74.106,Y -42.862,Z -63.398,A -90.000,B 90.000,C 0.000} C_DIS
LIN {X 74.743,Y -42.862,Z -62.055,A -90.000,B 90.000,C 0.000} C_DIS
LIN {X 75.432,Y -42.862,Z -60.738,A -90.000,B 90.000,C 0.000} C_DIS
LIN {X 76.171,Y -42.862,Z -59.448,A -90.000,B 90.000,C 0.000} C_DIS
LIN {X 76.961,Y -42.862,Z -58.189,A -90.000,B 90.000,C 0.000} C_DIS
LIN {X 77.798,Y -42.862,Z -56.961,A -90.000,B 90.000,C 0.000} C_DIS
LIN {X 78.683,Y -42.862,Z -55.767,A -90.000,B 90.000,C 0.000} C_DIS
LIN {X 79.921,Y -42.862,Z -54.319,A -90.000,B 90.000,C 0.000} C_DIS
LIN {X 81.197,Y -42.862,Z -52.905,A -90.000,B 90.000,C 0.000} C_DIS
LIN {X 82.511,Y -42.862,Z -51.525,A -90.000,B 90.000,C 0.000} C_DIS
LIN {X 83.862,Y -42.862,Z -50.182,A -90.000,B 90.000,C 0.000} C_DIS
LIN {X 85.248,Y -42.862,Z -48.875,A -90.000,B 90.000,C 0.000} C_DIS
LIN {X 86.669,Y -42.862,Z -47.605,A -90.000,B 90.000,C 0.000} C_DIS
LIN {X 88.123,Y -42.862,Z -46.375,A -90.000,B 90.000,C 0.000} C_DIS
LIN {X 89.414,Y -42.862,Z -45.330,A -90.000,B 90.000,C 0.000} C_DIS
LIN {X 90.669,Y -42.862,Z -44.241,A -90.000,B 90.000,C 0.000} C_DIS
LIN {X 91.885,Y -42.862,Z -43.110,A -90.000,B 90.000,C 0.000} C_DIS
LIN {X 93.063,Y -42.862,Z -41.938,A -90.000,B 90.000,C 0.000} C_DIS
LIN {X 94.200,Y -42.862,Z -40.727,A -90.000,B 90.000,C 0.000} C_DIS
LIN {X 95.405,Y -42.862,Z -39.283,A -90.000,B 90.000,C 0.000} C_DIS
LIN {X 96.652,Y -42.862,Z -37.876,A -90.000,B 90.000,C 0.000} C_DIS
LIN {X 97.940,Y -42.862,Z -36.505,A -90.000,B 90.000,C 0.000} C_DIS
LIN {X 99.268,Y -42.862,Z -35.173,A -90.000,B 90.000,C 0.000} C_DIS
LIN {X 100.634,Y -42.862,Z -33.880,A -90.000,B 90.000,C 0.000} C_DIS
LIN {X 102.037,Y -42.862,Z -32.628,A -90.000,B 90.000,C 0.000} C_DIS
LIN {X 102.777,Y -42.862,Z -32.024,A -90.000,B 90.000,C 0.000} C_DIS
LIN {X 103.556,Y -42.862,Z -31.472,A -90.000,B 90.000,C 0.000} C_DIS
LIN {X 104.372,Y -42.862,Z -30.975,A -90.000,B 90.000,C 0.000} C_DIS
LIN {X 105.220,Y -42.862,Z -30.536,A -90.000,B 90.000,C 0.000} C_DIS
LIN {X 106.097,Y -42.862,Z -30.157,A -90.000,B 90.000,C 0.000} C_DIS
LIN {X 106.998,Y -42.862,Z -29.840,A -90.000,B 90.000,C 0.000} C_DIS
LIN {X 107.918,Y -42.862,Z -29.585,A -90.000,B 90.000,C 0.000} C_DIS
LIN {X 108.854,Y -42.862,Z -29.395,A -90.000,B 90.000,C 0.000} C_DIS
LIN {X 109.801,Y -42.862,Z -29.270,A -90.000,B 90.000,C 0.000} C_DIS
LIN {X 110.755,Y -42.862,Z -29.210,A -90.000,B 90.000,C 0.000} C_DIS
LIN {X 111.710,Y -42.862,Z -29.217,A -90.000,B 90.000,C 0.000} C_DIS
LIN {X 112.662,Y -42.862,Z -29.290,A -90.000,B 90.000,C 0.000} C_DIS
LIN {X 112.818,Y -42.862,Z -29.320,A -90.000,B 90.000,C 0.000} C_DIS
LIN {X 112.905,Y -42.862,Z -29.324,A -90.000,B 90.000,C 0.000} C_DIS
LIN {X 113.833,Y -42.862,Z -29.470,A -90.000,B 90.000,C 0.000} C_DIS
LIN {X 114.748,Y -42.862,Z -29.684,A -90.000,B 90.000,C 0.000} C_DIS
LIN {X 115.644,Y -42.862,Z -29.965,A -90.000,B 90.000,C 0.000} C_DIS
LIN {X 116.518,Y -42.862,Z -30.312,A -90.000,B 90.000,C 0.000} C_DIS
LIN {X 117.363,Y -42.862,Z -30.721,A -90.000,B 90.000,C 0.000} C_DIS
LIN {X 118.176,Y -42.862,Z -31.192,A -90.000,B 90.000,C 0.000} C_DIS
LIN {X 118.952,Y -42.862,Z -31.722,A -90.000,B 90.000,C 0.000} C_DIS
LIN {X 119.687,Y -42.862,Z -32.307,A -90.000,B 90.000,C 0.000} C_DIS
LIN {X 120.377,Y -42.862,Z -32.945,A -90.000,B 90.000,C 0.000} C_DIS
LIN {X 121.018,Y -42.862,Z -33.632,A -90.000,B 90.000,C 0.000} C_DIS
LIN {X 121.607,Y -42.862,Z -34.364,A -90.000,B 90.000,C 0.000} C_DIS
LIN {X 122.140,Y -42.862,Z -35.138,A -90.000,B 90.000,C 0.000} C_DIS
LIN {X 122.615,Y -42.862,Z -35.949,A -90.000,B 90.000,C 0.000} C_DIS
LIN {X 123.028,Y -42.862,Z -36.792,A -90.000,B 90.000,C 0.000} C_DIS
LIN {X 123.379,Y -42.862,Z -37.664,A -90.000,B 90.000,C 0.000} C_DIS
LIN {X 123.664,Y -42.862,Z -38.559,A -90.000,B 90.000,C 0.000} C_DIS
LIN {X 123.709,Y -42.862,Z -38.736,A -90.000,B 90.000,C 0.000} C_DIS
LIN {X 123.902,Y -42.862,Z -39.558,A -90.000,B 90.000,C 0.000} C_DIS
LIN {X 124.042,Y -42.862,Z -40.390,A -90.000,B 90.000,C 0.000} C_DIS
LIN {X 124.128,Y -42.862,Z -41.230,A -90.000,B 90.000,C 0.000} C_DIS
LIN {X 124.160,Y -42.862,Z -42.074,A -90.000,B 90.000,C 0.000} C_DIS
LIN {X 124.137,Y -42.862,Z -42.918,A -90.000,B 90.000,C 0.000} C_DIS
LIN {X 123.900,Y -42.862,Z -44.315,A -90.000,B 90.000,C 0.000} C_DIS
LIN {X 123.599,Y -42.862,Z -45.700,A -90.000,B 90.000,C 0.000} C_DIS
LIN {X 123.236,Y -42.862,Z -47.070,A -90.000,B 90.000,C 0.000} C_DIS
LIN {X 122.811,Y -42.862,Z -48.422,A -90.000,B 90.000,C 0.000} C_DIS
LIN {X 122.324,Y -42.862,Z -49.753,A -90.000,B 90.000,C 0.000} C_DIS
LIN {X 121.777,Y -42.862,Z -51.060,A -90.000,B 90.000,C 0.000} C_DIS
LIN {X 120.906,Y -42.862,Z -52.689,A -90.000,B 90.000,C 0.000} C_DIS
LIN {X 120.085,Y -42.862,Z -54.344,A -90.000,B 90.000,C 0.000} C_DIS
LIN {X 119.315,Y -42.862,Z -56.022,A -90.000,B 90.000,C 0.000} C_DIS
LIN {X 118.595,Y -42.862,Z -57.723,A -90.000,B 90.000,C 0.000} C_DIS
LIN {X 117.927,Y -42.862,Z -59.445,A -90.000,B 90.000,C 0.000} C_DIS
LIN {X 117.105,Y -42.862,Z -62.047,A -90.000,B 90.000,C 0.000} C_DIS
LIN {X 116.236,Y -42.862,Z -64.633,A -90.000,B 90.000,C 0.000} C_DIS
LIN {X 115.318,Y -42.862,Z -67.203,A -90.000,B 90.000,C 0.000} C_DIS
LIN {X 114.353,Y -42.862,Z -69.755,A -90.000,B 90.000,C 0.000} C_DIS
LIN {X 113.342,Y -42.862,Z -72.289,A -90.000,B 90.000,C 0.000} C_DIS
LIN {X 112.640,Y -42.862,Z -74.060,A -90.000,B 90.000,C 0.000} C_DIS
LIN {X 111.875,Y -42.862,Z -75.805,A -90.000,B 90.000,C 0.000} C_DIS
LIN {X 111.050,Y -42.862,Z -77.522,A -90.000,B 90.000,C 0.000} C_DIS
LIN {X 110.164,Y -42.862,Z -79.209,A -90.000,B 90.000,C 0.000} C_DIS
LIN {X 109.220,Y -42.862,Z -80.863,A -90.000,B 90.000,C 0.000} C_DIS
LIN {X 108.218,Y -42.862,Z -82.484,A -90.000,B 90.000,C 0.000} C_DIS
LIN {X 107.159,Y -42.862,Z -84.068,A -90.000,B 90.000,C 0.000} C_DIS
LIN {X 106.045,Y -42.862,Z -85.613,A -90.000,B 90.000,C 0.000} C_DIS
LIN {X 105.204,Y -42.862,Z -86.770,A -90.000,B 90.000,C 0.000} C_DIS
LIN {X 104.309,Y -42.862,Z -87.886,A -90.000,B 90.000,C 0.000} C_DIS
LIN {X 103.362,Y -42.862,Z -88.959,A -90.000,B 90.000,C 0.000} C_DIS
LIN {X 102.367,Y -42.862,Z -89.986,A -90.000,B 90.000,C 0.000} C_DIS
LIN {X 101.324,Y -42.862,Z -90.965,A -90.000,B 90.000,C 0.000} C_DIS
LIN {X 100.236,Y -42.862,Z -91.894,A -90.000,B 90.000,C 0.000} C_DIS
LIN {X 99.106,Y -42.862,Z -92.771,A -90.000,B 90.000,C 0.000} C_DIS
LIN {X 98.992,Y -42.862,Z -94.148,A -90.000,B 90.000,C 0.000} C_DIS
LIN {X 98.825,Y -42.862,Z -95.520,A -90.000,B 90.000,C 0.000} C_DIS
LIN {X 98.608,Y -42.862,Z -96.884,A -90.000,B 90.000,C 0.000} C_DIS
LIN {X 98.338,Y -42.862,Z -98.239,A -90.000,B 90.000,C 0.000} C_DIS
LIN {X 98.104,Y -42.862,Z -99.170,A -90.000,B 90.000,C 0.000} C_DIS
LIN {X 97.807,Y -42.862,Z -100.084,A -90.000,B 90.000,C 0.000} C_DIS
LIN {X 97.448,Y -42.862,Z -100.974,A -90.000,B 90.000,C 0.000} C_DIS
LIN {X 97.029,Y -42.862,Z -101.839,A -90.000,B 90.000,C 0.000} C_DIS
LIN {X 96.552,Y -42.862,Z -102.672,A -90.000,B 90.000,C 0.000} C_DIS
LIN {X 96.020,Y -42.862,Z -103.472,A -90.000,B 90.000,C 0.000} C_DIS
LIN {X 95.434,Y -42.862,Z -104.233,A -90.000,B 90.000,C 0.000} C_DIS
LIN {X 94.798,Y -42.862,Z -104.952,A -90.000,B 90.000,C 0.000} C_DIS
LIN {X 94.904,Y -42.862,Z -106.052,A -90.000,B 90.000,C 0.000} C_DIS
LIN {X 94.961,Y -42.862,Z -107.157,A -90.000,B 90.000,C 0.000} C_DIS
LIN {X 94.968,Y -42.862,Z -108.262,A -90.000,B 90.000,C 0.000} C_DIS
LIN {X 94.801,Y -42.862,Z -109.804,A -90.000,B 90.000,C 0.000} C_DIS
LIN {X 94.574,Y -42.862,Z -111.338,A -90.000,B 90.000,C 0.000} C_DIS
LIN {X 94.286,Y -42.862,Z -112.862,A -90.000,B 90.000,C 0.000} C_DIS
LIN {X 93.940,Y -42.862,Z -114.373,A -90.000,B 90.000,C 0.000} C_DIS
LIN {X 93.534,Y -42.862,Z -115.870,A -90.000,B 90.000,C 0.000} C_DIS
LIN {X 93.163,Y -42.862,Z -116.870,A -90.000,B 90.000,C 0.000} C_DIS
LIN {X 92.830,Y -42.862,Z -117.883,A -90.000,B 90.000,C 0.000} C_DIS
LIN {X 92.536,Y -42.862,Z -118.908,A -90.000,B 90.000,C 0.000} C_DIS
LIN {X 92.535,Y -42.862,Z -119.054,A -90.000,B 90.000,C 0.000} C_DIS
LIN {X 92.689,Y -42.862,Z -120.067,A -90.000,B 90.000,C 0.000} C_DIS
LIN {X 92.875,Y -42.862,Z -121.074,A -90.000,B 90.000,C 0.000} C_DIS
LIN {X 93.094,Y -42.862,Z -122.075,A -90.000,B 90.000,C 0.000} C_DIS
LIN {X 93.300,Y -42.862,Z -123.753,A -90.000,B 90.000,C 0.000} C_DIS
LIN {X 93.441,Y -42.862,Z -125.438,A -90.000,B 90.000,C 0.000} C_DIS
LIN {X 93.516,Y -42.862,Z -127.127,A -90.000,B 90.000,C 0.000} C_DIS
LIN {X 93.526,Y -42.862,Z -128.817,A -90.000,B 90.000,C 0.000} C_DIS
LIN {X 93.471,Y -42.862,Z -130.507,A -90.000,B 90.000,C 0.000} C_DIS
LIN {X 93.350,Y -42.862,Z -132.193,A -90.000,B 90.000,C 0.000} C_DIS
LIN {X 93.075,Y -42.862,Z -138.416,A -90.000,B 90.000,C 0.000} C_DIS
LIN {X 92.760,Y -42.862,Z -144.638,A -90.000,B 90.000,C 0.000} C_DIS
LIN {X 92.614,Y -42.862,Z -147.160,A -90.000,B 90.000,C 0.000} C_DIS
LIN {X 92.407,Y -42.862,Z -149.677,A -90.000,B 90.000,C 0.000} C_DIS
LIN {X 92.139,Y -42.862,Z -152.188,A -90.000,B 90.000,C 0.000} C_DIS
LIN {X 91.809,Y -42.862,Z -154.692,A -90.000,B 90.000,C 0.000} C_DIS
LIN {X 91.418,Y -42.862,Z -157.188,A -90.000,B 90.000,C 0.000} C_DIS
LIN {X 90.966,Y -42.862,Z -159.673,A -90.000,B 90.000,C 0.000} C_DIS
LIN {X 90.454,Y -42.862,Z -162.146,A -90.000,B 90.000,C 0.000} C_DIS
LIN {X 89.881,Y -42.862,Z -164.606,A -90.000,B 90.000,C 0.000} C_DIS
LIN {X 89.249,Y -42.862,Z -167.051,A -90.000,B 90.000,C 0.000} C_DIS
LIN {X 88.557,Y -42.862,Z -169.480,A -90.000,B 90.000,C 0.000} C_DIS
LIN {X 87.806,Y -42.862,Z -171.892,A -90.000,B 90.000,C 0.000} C_DIS
LIN {X 86.713,Y -42.862,Z -175.316,A -90.000,B 90.000,C 0.000} C_DIS
LIN {X 85.641,Y -42.862,Z -178.746,A -90.000,B 90.000,C 0.000} C_DIS
LIN {X 84.339,Y -42.862,Z -184.045,A -90.000,B 90.000,C 0.000} C_DIS
LIN {X 82.986,Y -42.862,Z -189.331,A -90.000,B 90.000,C 0.000} C_DIS
LIN {X 81.580,Y -42.862,Z -194.604,A -90.000,B 90.000,C 0.000} C_DIS
LIN {X 80.215,Y -42.862,Z -198.706,A -90.000,B 90.000,C 0.000} C_DIS
LIN {X 78.786,Y -42.862,Z -202.786,A -90.000,B 90.000,C 0.000} C_DIS
LIN {X 77.296,Y -42.862,Z -206.844,A -90.000,B 90.000,C 0.000} C_DIS
LIN {X 75.743,Y -42.862,Z -210.878,A -90.000,B 90.000,C 0.000} C_DIS
LIN {X 74.128,Y -42.862,Z -214.888,A -90.000,B 90.000,C 0.000} C_DIS
LIN {X 72.452,Y -42.862,Z -218.873,A -90.000,B 90.000,C 0.000} C_DIS
LIN {X 70.715,Y -42.862,Z -222.832,A -90.000,B 90.000,C 0.000} C_DIS
LIN {X 68.918,Y -42.862,Z -226.763,A -90.000,B 90.000,C 0.000} C_DIS
LIN {X 67.060,Y -42.862,Z -230.667,A -90.000,B 90.000,C 0.000} C_DIS
LIN {X 65.797,Y -42.862,Z -233.305,A -90.000,B 90.000,C 0.000} C_DIS
LIN {X 64.477,Y -42.862,Z -235.915,A -90.000,B 90.000,C 0.000} C_DIS
LIN {X 63.099,Y -42.862,Z -238.495,A -90.000,B 90.000,C 0.000} C_DIS
LIN {X 61.666,Y -42.862,Z -241.044,A -90.000,B 90.000,C 0.000} C_DIS
LIN {X 60.176,Y -42.862,Z -243.561,A -90.000,B 90.000,C 0.000} C_DIS
LIN {X 145.015,Y -42.862,Z -243.561,A -90.000,B 90.000,C 0.000} C_DIS
LIN {X 145.015,Y -42.862,Z 0.000,A -90.000,B 90.000,C 0.000} C_DIS
LIN {X -145.015,Y -42.862,Z 0.000,A -90.000,B 90.000,C 0.000} C_DIS
LIN {X -145.015,Y -42.862,Z -243.561,A -90.000,B 90.000,C 0.000} C_DIS
LIN {X -95.683,Y -42.862,Z -243.561,A -90.000,B 90.000,C 0.000} C_DIS
LIN {X -93.388,Y -42.862,Z -241.976,A -90.000,B 90.000,C 0.000} C_DIS
LIN {X -91.062,Y -42.862,Z -240.436,A -90.000,B 90.000,C 0.000} C_DIS
LIN {X -88.708,Y -42.862,Z -238.941,A -90.000,B 90.000,C 0.000} C_DIS
LIN {X -86.326,Y -42.862,Z -237.490,A -90.000,B 90.000,C 0.000} C_DIS
LIN {X -81.927,Y -42.862,Z -234.928,A -90.000,B 90.000,C 0.000} C_DIS
LIN {X -77.499,Y -42.862,Z -232.415,A -90.000,B 90.000,C 0.000} C_DIS
LIN {X -73.043,Y -42.862,Z -229.952,A -90.000,B 90.000,C 0.000} C_DIS
LIN {X -68.559,Y -42.862,Z -227.539,A -90.000,B 90.000,C 0.000} C_DIS
LIN {X -64.049,Y -42.862,Z -225.177,A -90.000,B 90.000,C 0.000} C_DIS
LIN {X -59.513,Y -42.862,Z -222.865,A -90.000,B 90.000,C 0.000} C_DIS
LIN {X -54.951,Y -42.862,Z -220.605,A -90.000,B 90.000,C 0.000} C_DIS
LIN {X -47.202,Y -42.862,Z -216.835,A -90.000,B 90.000,C 0.000} C_DIS
LIN {X -43.562,Y -42.862,Z -215.185,A -90.000,B 90.000,C 0.000} C_DIS
LIN {X -39.942,Y -42.862,Z -213.491,A -90.000,B 90.000,C 0.000} C_DIS
LIN {X -36.344,Y -42.862,Z -211.752,A -90.000,B 90.000,C 0.000} C_DIS
LIN {X -32.767,Y -42.862,Z -209.968,A -90.000,B 90.000,C 0.000} C_DIS
LIN {X -30.475,Y -42.862,Z -208.934,A -90.000,B 90.000,C 0.000} C_DIS
LIN {X -28.210,Y -42.862,Z -207.841,A -90.000,B 90.000,C 0.000} C_DIS
LIN {X -25.975,Y -42.862,Z -206.690,A -90.000,B 90.000,C 0.000} C_DIS
LIN {X -23.770,Y -42.862,Z -205.481,A -90.000,B 90.000,C 0.000} C_DIS
LIN {X -21.598,Y -42.862,Z -204.214,A -90.000,B 90.000,C 0.000} C_DIS
LIN {X -19.459,Y -42.862,Z -202.892,A -90.000,B 90.000,C 0.000} C_DIS
LIN {X -17.332,Y -42.862,Z -201.616,A -90.000,B 90.000,C 0.000} C_DIS
LIN {X -15.240,Y -42.862,Z -200.285,A -90.000,B 90.000,C 0.000} C_DIS
LIN {X -13.182,Y -42.862,Z -198.900,A -90.000,B 90.000,C 0.000} C_DIS
LIN {X -11.161,Y -42.862,Z -197.463,A -90.000,B 90.000,C 0.000} C_DIS
LIN {X -9.178,Y -42.862,Z -195.973,A -90.000,B 90.000,C 0.000} C_DIS
LIN {X -7.234,Y -42.862,Z -194.432,A -90.000,B 90.000,C 0.000} C_DIS
LIN {X -5.331,Y -42.862,Z -192.842,A -90.000,B 90.000,C 0.000} C_DIS
LIN {X -3.470,Y -42.862,Z -191.203,A -90.000,B 90.000,C 0.000} C_DIS
LIN {X -1.652,Y -42.862,Z -189.516,A -90.000,B 90.000,C 0.000} C_DIS
LIN {X 0.121,Y -42.862,Z -187.782,A -90.000,B 90.000,C 0.000} C_DIS
LIN {X 1.849,Y -42.862,Z -186.003,A -90.000,B 90.000,C 0.000} C_DIS
LIN {X 3.531,Y -42.862,Z -184.180,A -90.000,B 90.000,C 0.000} C_DIS
LIN {X 5.269,Y -42.862,Z -182.176,A -90.000,B 90.000,C 0.000} C_DIS
LIN {X 7.041,Y -42.862,Z -180.202,A -90.000,B 90.000,C 0.000} C_DIS
LIN {X 8.848,Y -42.862,Z -178.260,A -90.000,B 90.000,C 0.000} C_DIS
LIN {X 10.689,Y -42.862,Z -176.350,A -90.000,B 90.000,C 0.000} C_DIS
LIN {X 12.563,Y -42.862,Z -174.472,A -90.000,B 90.000,C 0.000} C_DIS
LIN {X 14.470,Y -42.862,Z -172.628,A -90.000,B 90.000,C 0.000} C_DIS
LIN {X 15.782,Y -42.862,Z -171.493,A -90.000,B 90.000,C 0.000} C_DIS
LIN {X 17.051,Y -42.862,Z -170.309,A -90.000,B 90.000,C 0.000} C_DIS
LIN {X 18.276,Y -42.862,Z -169.080,A -90.000,B 90.000,C 0.000} C_DIS
LIN {X 19.453,Y -42.862,Z -167.806,A -90.000,B 90.000,C 0.000} C_DIS
LIN {X 20.583,Y -42.862,Z -166.489,A -90.000,B 90.000,C 0.000} C_DIS
LIN {X 21.664,Y -42.862,Z -165.131,A -90.000,B 90.000,C 0.000} C_DIS
LIN {X 22.693,Y -42.862,Z -163.734,A -90.000,B 90.000,C 0.000} C_DIS
LIN {X 23.669,Y -42.862,Z -162.300,A -90.000,B 90.000,C 0.000} C_DIS
LIN {X 24.637,Y -42.862,Z -160.908,A -90.000,B 90.000,C 0.000} C_DIS
LIN {X 25.552,Y -42.862,Z -159.481,A -90.000,B 90.000,C 0.000} C_DIS
LIN {X 26.415,Y -42.862,Z -158.022,A -90.000,B 90.000,C 0.000} C_DIS
LIN {X 27.224,Y -42.862,Z -156.532,A -90.000,B 90.000,C 0.000} C_DIS
LIN {X 27.978,Y -42.862,Z -155.014,A -90.000,B 90.000,C 0.000} C_DIS
LIN {X 28.676,Y -42.862,Z -153.469,A -90.000,B 90.000,C 0.000} C_DIS
LIN {X 29.316,Y -42.862,Z -151.899,A -90.000,B 90.000,C 0.000} C_DIS
LIN {X 29.899,Y -42.862,Z -150.307,A -90.000,B 90.000,C 0.000} C_DIS
LIN {X 29.982,Y -42.862,Z -150.108,A -90.000,B 90.000,C 0.000} C_DIS
LIN {X 26.378,Y -42.862,Z -152.030,A -90.000,B 90.000,C 0.000} C_DIS
LIN {X 24.481,Y -42.862,Z -152.881,A -90.000,B 90.000,C 0.000} C_DIS
LIN {X 22.555,Y -42.862,Z -153.667,A -90.000,B 90.000,C 0.000} C_DIS
LIN {X 20.605,Y -42.862,Z -154.387,A -90.000,B 90.000,C 0.000} C_DIS
LIN {X 18.630,Y -42.862,Z -155.040,A -90.000,B 90.000,C 0.000} C_DIS
LIN {X 16.635,Y -42.862,Z -155.626,A -90.000,B 90.000,C 0.000} C_DIS
LIN {X 14.621,Y -42.862,Z -156.143,A -90.000,B 90.000,C 0.000} C_DIS
LIN {X 12.591,Y -42.862,Z -156.592,A -90.000,B 90.000,C 0.000} C_DIS
LIN {X 10.546,Y -42.862,Z -156.971,A -90.000,B 90.000,C 0.000} C_DIS
LIN {X 8.490,Y -42.862,Z -157.281,A -90.000,B 90.000,C 0.000} C_DIS
LIN {X 6.424,Y -42.862,Z -157.520,A -90.000,B 90.000,C 0.000} C_DIS
LIN {X 4.796,Y -42.862,Z -157.590,A -90.000,B 90.000,C 0.000} C_DIS
LIN {X 3.167,Y -42.862,Z -157.596,A -90.000,B 90.000,C 0.000} C_DIS
LIN {X 1.538,Y -42.862,Z -157.540,A -90.000,B 90.000,C 0.000} C_DIS
LIN {X -0.087,Y -42.862,Z -157.420,A -90.000,B 90.000,C 0.000} C_DIS
LIN {X -1.706,Y -42.862,Z -157.238,A -90.000,B 90.000,C 0.000} C_DIS
LIN {X -3.317,Y -42.862,Z -156.994,A -90.000,B 90.000,C 0.000} C_DIS
LIN {X -4.917,Y -42.862,Z -156.687,A -90.000,B 90.000,C 0.000} C_DIS
LIN {X -6.504,Y -42.862,Z -156.319,A -90.000,B 90.000,C 0.000} C_DIS
LIN {X -8.076,Y -42.862,Z -155.890,A -90.000,B 90.000,C 0.000} C_DIS
LIN {X -9.630,Y -42.862,Z -155.400,A -90.000,B 90.000,C 0.000} C_DIS
LIN {X -11.164,Y -42.862,Z -154.851,A -90.000,B 90.000,C 0.000} C_DIS
LIN {X -12.676,Y -42.862,Z -154.243,A -90.000,B 90.000,C 0.000} C_DIS
LIN {X -14.163,Y -42.862,Z -153.577,A -90.000,B 90.000,C 0.000} C_DIS
LIN {X -15.690,Y -42.862,Z -152.777,A -90.000,B 90.000,C 0.000} C_DIS
LIN {X -17.188,Y -42.862,Z -151.923,A -90.000,B 90.000,C 0.000} C_DIS
LIN {X -18.655,Y -42.862,Z -151.018,A -90.000,B 90.000,C 0.000} C_DIS
LIN {X -20.089,Y -42.862,Z -150.062,A -90.000,B 90.000,C 0.000} C_DIS
LIN {X -21.489,Y -42.862,Z -149.056,A -90.000,B 90.000,C 0.000} C_DIS
LIN {X -22.852,Y -42.862,Z -148.001,A -90.000,B 90.000,C 0.000} C_DIS
LIN {X -24.178,Y -42.862,Z -146.899,A -90.000,B 90.000,C 0.000} C_DIS
LIN {X -25.464,Y -42.862,Z -145.752,A -90.000,B 90.000,C 0.000} C_DIS
LIN {X -26.709,Y -42.862,Z -144.559,A -90.000,B 90.000,C 0.000} C_DIS
LIN {X -27.819,Y -42.862,Z -143.291,A -90.000,B 90.000,C 0.000} C_DIS
LIN {X -28.875,Y -42.862,Z -141.978,A -90.000,B 90.000,C 0.000} C_DIS
LIN {X -29.876,Y -42.862,Z -140.623,A -90.000,B 90.000,C 0.000} C_DIS
LIN {X -30.819,Y -42.862,Z -139.226,A -90.000,B 90.000,C 0.000} C_DIS
LIN {X -31.704,Y -42.862,Z -137.792,A -90.000,B 90.000,C 0.000} C_DIS
LIN {X -32.527,Y -42.862,Z -136.322,A -90.000,B 90.000,C 0.000} C_DIS
LIN {X -33.290,Y -42.862,Z -134.819,A -90.000,B 90.000,C 0.000} C_DIS
LIN {X -33.988,Y -42.862,Z -133.286,A -90.000,B 90.000,C 0.000} C_DIS
LIN {X -34.623,Y -42.862,Z -131.725,A -90.000,B 90.000,C 0.000} C_DIS
LIN {X -35.192,Y -42.862,Z -130.139,A -90.000,B 90.000,C 0.000} C_DIS
LIN {X -35.611,Y -42.862,Z -129.333,A -90.000,B 90.000,C 0.000} C_DIS
LIN {X -35.977,Y -42.862,Z -128.503,A -90.000,B 90.000,C 0.000} C_DIS
LIN {X -36.289,Y -42.862,Z -127.650,A -90.000,B 90.000,C 0.000} C_DIS
LIN {X -36.545,Y -42.862,Z -126.779,A -90.000,B 90.000,C 0.000} C_DIS
LIN {X -36.965,Y -42.862,Z -125.741,A -90.000,B 90.000,C 0.000} C_DIS
LIN {X -37.354,Y -42.862,Z -124.692,A -90.000,B 90.000,C 0.000} C_DIS
LIN {X -37.714,Y -42.862,Z -123.633,A -90.000,B 90.000,C 0.000} C_DIS
LIN {X -38.044,Y -42.862,Z -122.563,A -90.000,B 90.000,C 0.000} C_DIS
LIN {X -38.429,Y -42.862,Z -121.536,A -90.000,B 90.000,C 0.000} C_DIS
LIN {X -38.782,Y -42.862,Z -120.498,A -90.000,B 90.000,C 0.000} C_DIS
LIN {X -39.104,Y -42.862,Z -119.450,A -90.000,B 90.000,C 0.000} C_DIS
LIN {X -39.134,Y -42.862,Z -119.293,A -90.000,B 90.000,C 0.000} C_DIS
LIN {X -39.186,Y -42.862,Z -119.113,A -90.000,B 90.000,C 0.000} C_DIS
LIN {X -39.644,Y -42.862,Z -116.929,A -90.000,B 90.000,C 0.000} C_DIS
LIN {X -40.135,Y -42.862,Z -114.753,A -90.000,B 90.000,C 0.000} C_DIS
LIN {X -40.301,Y -42.862,Z -112.993,A -90.000,B 90.000,C 0.000} C_DIS
LIN {X -40.426,Y -42.862,Z -111.230,A -90.000,B 90.000,C 0.000} C_DIS
LIN {X -40.509,Y -42.862,Z -109.464,A -90.000,B 90.000,C 0.000} C_DIS
LIN {X -40.551,Y -42.862,Z -107.697,A -90.000,B 90.000,C 0.000} C_DIS
LIN {X -40.347,Y -42.862,Z -105.682,A -90.000,B 90.000,C 0.000} C_DIS
LIN {X -40.090,Y -42.862,Z -103.672,A -90.000,B 90.000,C 0.000} C_DIS
LIN {X -39.780,Y -42.862,Z -101.670,A -90.000,B 90.000,C 0.000} C_DIS
LIN {X -39.417,Y -42.862,Z -99.677,A -90.000,B 90.000,C 0.000} C_DIS
LIN {X -39.001,Y -42.862,Z -97.695,A -90.000,B 90.000,C 0.000} C_DIS
LIN {X -38.532,Y -42.862,Z -95.724,A -90.000,B 90.000,C 0.000} C_DIS
LIN {X -38.012,Y -42.862,Z -93.766,A -90.000,B 90.000,C 0.000} C_DIS
LIN {X -37.452,Y -42.862,Z -92.152,A -90.000,B 90.000,C 0.000} C_DIS
LIN {X -36.832,Y -42.862,Z -90.561,A -90.000,B 90.000,C 0.000} C_DIS
LIN {X -36.152,Y -42.862,Z -88.994,A -90.000,B 90.000,C 0.000} C_DIS
LIN {X -35.414,Y -42.862,Z -87.453,A -90.000,B 90.000,C 0.000} C_DIS
LIN {X -34.618,Y -42.862,Z -85.942,A -90.000,B 90.000,C 0.000} C_DIS
LIN {X -33.766,Y -42.862,Z -84.462,A -90.000,B 90.000,C 0.000} C_DIS
LIN {X -32.859,Y -42.862,Z -83.014,A -90.000,B 90.000,C 0.000} C_DIS
LIN {X -31.897,Y -42.862,Z -81.602,A -90.000,B 90.000,C 0.000} C_DIS
LIN {X -30.884,Y -42.862,Z -80.227,A -90.000,B 90.000,C 0.000} C_DIS
LIN {X -29.819,Y -42.862,Z -78.892,A -90.000,B 90.000,C 0.000} C_DIS
LIN {X -28.705,Y -42.862,Z -77.597,A -90.000,B 90.000,C 0.000} C_DIS
LIN {X -27.899,Y -42.862,Z -76.674,A -90.000,B 90.000,C 0.000} C_DIS
LIN {X -27.043,Y -42.862,Z -75.797,A -90.000,B 90.000,C 0.000} C_DIS
LIN {X -26.142,Y -42.862,Z -74.966,A -90.000,B 90.000,C 0.000} C_DIS
LIN {X -25.198,Y -42.862,Z -74.186,A -90.000,B 90.000,C 0.000} C_DIS
LIN {X -24.212,Y -42.862,Z -73.458,A -90.000,B 90.000,C 0.000} C_DIS
LIN {X -23.189,Y -42.862,Z -72.784,A -90.000,B 90.000,C 0.000} C_DIS
LIN {X -22.131,Y -42.862,Z -72.166,A -90.000,B 90.000,C 0.000} C_DIS
LIN {X -21.041,Y -42.862,Z -71.606,A -90.000,B 90.000,C 0.000} C_DIS
LIN {X -19.922,Y -42.862,Z -71.106,A -90.000,B 90.000,C 0.000} C_DIS
LIN {X -18.778,Y -42.862,Z -70.667,A -90.000,B 90.000,C 0.000} C_DIS
LIN {X -17.612,Y -42.862,Z -70.290,A -90.000,B 90.000,C 0.000} C_DIS
LIN {X -16.427,Y -42.862,Z -69.977,A -90.000,B 90.000,C 0.000} C_DIS
LIN {X -15.227,Y -42.862,Z -69.728,A -90.000,B 90.000,C 0.000} C_DIS
LIN {X -14.016,Y -42.862,Z -69.544,A -90.000,B 90.000,C 0.000} C_DIS
LIN {X -12.796,Y -42.862,Z -69.426,A -90.000,B 90.000,C 0.000} C_DIS
LIN {X -11.755,Y -42.862,Z -69.310,A -90.000,B 90.000,C 0.000} C_DIS
LIN {X -10.709,Y -42.862,Z -69.250,A -90.000,B 90.000,C 0.000} C_DIS
LIN {X -9.661,Y -42.862,Z -69.246,A -90.000,B 90.000,C 0.000} C_DIS
LIN {X -8.615,Y -42.862,Z -69.299,A -90.000,B 90.000,C 0.000} C_DIS
LIN {X -7.573,Y -42.862,Z -69.409,A -90.000,B 90.000,C 0.000} C_DIS
LIN {X -7.573,Y -55.362,Z -69.409,A -90.000,B 90.000,C 0.000} C_DIS
LIN {X -7.573,Y -67.862,Z -69.409,A -90.000,B 90.000,C 0.000} C_DIS
LIN {X -110.443,Y -67.862,Z -242.561,A -90.000,B 90.000,C 0.000} C_DIS
LIN {X -110.443,Y -60.719,Z -242.561,A -90.000,B 90.000,C 0.000} C_DIS
LIN {X -110.443,Y -48.219,Z -242.561,A -90.000,B 90.000,C 0.000} C_DIS
LIN {X -110.443,Y -35.719,Z -242.561,A -90.000,B 90.000,C 0.000} C_DIS
LIN {X -144.015,Y -35.719,Z -242.561,A -90.000,B 90.000,C 0.000} C_DIS
LIN {X -144.015,Y -35.719,Z -235.012,A -90.000,B 90.000,C 0.000} C_DIS
LIN {X -100.345,Y -35.719,Z -235.012,A -90.000,B 90.000,C 0.000} C_DIS
LIN {X -97.633,Y -35.719,Z -233.116,A -90.000,B 90.000,C 0.000} C_DIS
LIN {X -94.895,Y -35.719,Z -231.255,A -90.000,B 90.000,C 0.000} C_DIS
LIN {X -92.134,Y -35.719,Z -229.431,A -90.000,B 90.000,C 0.000} C_DIS
LIN {X -89.348,Y -35.719,Z -227.645,A -90.000,B 90.000,C 0.000} C_DIS
LIN {X -89.073,Y -35.719,Z -227.464,A -90.000,B 90.000,C 0.000} C_DIS
LIN {X -144.015,Y -35.719,Z -227.464,A -90.000,B 90.000,C 0.000} C_DIS
LIN {X -144.015,Y -35.719,Z -219.915,A -90.000,B 90.000,C 0.000} C_DIS
LIN {X -76.577,Y -35.719,Z -219.915,A -90.000,B 90.000,C 0.000} C_DIS
LIN {X -73.135,Y -35.719,Z -217.973,A -90.000,B 90.000,C 0.000} C_DIS
LIN {X -69.672,Y -35.719,Z -216.068,A -90.000,B 90.000,C 0.000} C_DIS
LIN {X -66.190,Y -35.719,Z -214.199,A -90.000,B 90.000,C 0.000} C_DIS
LIN {X -62.688,Y -35.719,Z -212.366,A -90.000,B 90.000,C 0.000} C_DIS
LIN {X -144.015,Y -35.719,Z -212.366,A -90.000,B 90.000,C 0.000} C_DIS
LIN {X -144.015,Y -35.719,Z -204.817,A -90.000,B 90.000,C 0.000} C_DIS
LIN {X -47.545,Y -35.719,Z -204.817,A -90.000,B 90.000,C 0.000} C_DIS
LIN {X -47.374,Y -35.719,Z -204.732,A -90.000,B 90.000,C 0.000} C_DIS
LIN {X -45.022,Y -35.719,Z -203.596,A -90.000,B 90.000,C 0.000} C_DIS
LIN {X -42.692,Y -35.719,Z -202.416,A -90.000,B 90.000,C 0.000} C_DIS
LIN {X -40.384,Y -35.719,Z -201.193,A -90.000,B 90.000,C 0.000} C_DIS
LIN {X -38.100,Y -35.719,Z -199.927,A -90.000,B 90.000,C 0.000} C_DIS
LIN {X -35.839,Y -35.719,Z -198.619,A -90.000,B 90.000,C 0.000} C_DIS
LIN {X -33.603,Y -35.719,Z -197.269,A -90.000,B 90.000,C 0.000} C_DIS
LIN {X -144.015,Y -35.719,Z -197.269,A -90.000,B 90.000,C 0.000} C_DIS
LIN {X -144.015,Y -35.719,Z -189.720,A -90.000,B 90.000,C 0.000} C_DIS
LIN {X -22.799,Y -35.719,Z -189.720,A -90.000,B 90.000,C 0.000} C_DIS
LIN {X -20.437,Y -35.719,Z -187.878,A -90.000,B 90.000,C 0.000} C_DIS
LIN {X -18.098,Y -35.719,Z -186.006,A -90.000,B 90.000,C 0.000} C_DIS
LIN {X -15.784,Y -35.719,Z -184.103,A -90.000,B 90.000,C 0.000} C_DIS
LIN {X -13.495,Y -35.719,Z -182.171,A -90.000,B 90.000,C 0.000} C_DIS
LIN {X -144.015,Y -35.719,Z -182.171,A -90.000,B 90.000,C 0.000} C_DIS
LIN {X -144.015,Y -35.719,Z -174.622,A -90.000,B 90.000,C 0.000} C_DIS
LIN {X -4.987,Y -35.719,Z -174.622,A -90.000,B 90.000,C 0.000} C_DIS
LIN {X -3.657,Y -35.719,Z -173.349,A -90.000,B 90.000,C 0.000} C_DIS
LIN {X -2.350,Y -35.719,Z -172.053,A -90.000,B 90.000,C 0.000} C_DIS
LIN {X -1.066,Y -35.719,Z -170.733,A -90.000,B 90.000,C 0.000} C_DIS
LIN {X 0.193,Y -35.719,Z -169.390,A -90.000,B 90.000,C 0.000} C_DIS
LIN {X 0.701,Y -35.719,Z -168.856,A -90.000,B 90.000,C 0.000} C_DIS
LIN {X 1.175,Y -35.719,Z -168.290,A -90.000,B 90.000,C 0.000} C_DIS
LIN {X 1.610,Y -35.719,Z -167.695,A -90.000,B 90.000,C 0.000} C_DIS
LIN {X 2.007,Y -35.719,Z -167.073,A -90.000,B 90.000,C 0.000} C_DIS
LIN {X -144.015,Y -35.719,Z -167.073,A -90.000,B 90.000,C 0.000} C_DIS
LIN {X -144.015,Y -35.719,Z -159.525,A -90.000,B 90.000,C 0.000} C_DIS
LIN {X -12.789,Y -35.719,Z -159.525,A -90.000,B 90.000,C 0.000} C_DIS
LIN {X -14.386,Y -35.719,Z -158.767,A -90.000,B 90.000,C 0.000} C_DIS
LIN {X -15.968,Y -35.719,Z -157.977,A -90.000,B 90.000,C 0.000} C_DIS
LIN {X -17.534,Y -35.719,Z -157.158,A -90.000,B 90.000,C 0.000} C_DIS
LIN {X -19.084,Y -35.719,Z -156.307,A -90.000,B 90.000,C 0.000} C_DIS
LIN {X -21.256,Y -35.719,Z -154.904,A -90.000,B 90.000,C 0.000} C_DIS
LIN {X -23.402,Y -35.719,Z -153.460,A -90.000,B 90.000,C 0.000} C_DIS
LIN {X -25.519,Y -35.719,Z -151.976,A -90.000,B 90.000,C 0.000} C_DIS
LIN {X -144.015,Y -35.719,Z -151.976,A -90.000,B 90.000,C 0.000} C_DIS
LIN {X -144.015,Y -35.719,Z -144.427,A -90.000,B 90.000,C 0.000} C_DIS
LIN {X -34.320,Y -35.719,Z -144.427,A -90.000,B 90.000,C 0.000} C_DIS
LIN {X -35.446,Y -35.719,Z -143.258,A -90.000,B 90.000,C 0.000} C_DIS
LIN {X -36.532,Y -35.719,Z -142.051,A -90.000,B 90.000,C 0.000} C_DIS
LIN {X -37.576,Y -35.719,Z -140.808,A -90.000,B 90.000,C 0.000} C_DIS
LIN {X -38.578,Y -35.719,Z -139.531,A -90.000,B 90.000,C 0.000} C_DIS
LIN {X -39.536,Y -35.719,Z -138.220,A -90.000,B 90.000,C 0.000} C_DIS
LIN {X -40.449,Y -35.719,Z -136.878,A -90.000,B 90.000,C 0.000} C_DIS
LIN {X -144.015,Y -35.719,Z -136.878,A -90.000,B 90.000,C 0.000} C_DIS
LIN {X -144.015,Y -35.719,Z -129.329,A -90.000,B 90.000,C 0.000} C_DIS
LIN {X -44.485,Y -35.719,Z -129.329,A -90.000,B 90.000,C 0.000} C_DIS
LIN {X -45.083,Y -35.719,Z -127.854,A -90.000,B 90.000,C 0.000} C_DIS
LIN {X -45.631,Y -35.719,Z -126.360,A -90.000,B 90.000,C 0.000} C_DIS
LIN {X -46.130,Y -35.719,Z -124.849,A -90.000,B 90.000,C 0.000} C_DIS
LIN {X -46.578,Y -35.719,Z -123.322,A -90.000,B 90.000,C 0.000} C_DIS
LIN {X -46.976,Y -35.719,Z -121.781,A -90.000,B 90.000,C 0.000} C_DIS
LIN {X -144.015,Y -35.719,Z -121.781,A -90.000,B 90.000,C 0.000} C_DIS
LIN {X -144.015,Y -35.719,Z -114.232,A -90.000,B 90.000,C 0.000} C_DIS
LIN {X -48.192,Y -35.719,Z -114.232,A -90.000,B 90.000,C 0.000} C_DIS
LIN {X -48.332,Y -35.719,Z -112.748,A -90.000,B 90.000,C 0.000} C_DIS
LIN {X -48.440,Y -35.719,Z -111.261,A -90.000,B 90.000,C 0.000} C_DIS
LIN {X -48.517,Y -35.719,Z -109.772,A -90.000,B 90.000,C 0.000} C_DIS
LIN {X -48.869,Y -35.719,Z -109.262,A -90.000,B 90.000,C 0.000} C_DIS
LIN {X -49.245,Y -35.719,Z -108.770,A -90.000,B 90.000,C 0.000} C_DIS
LIN {X -49.644,Y -35.719,Z -108.296,A -90.000,B 90.000,C 0.000} C_DIS
LIN {X -50.292,Y -35.719,Z -107.496,A -90.000,B 90.000,C 0.000} C_DIS
LIN {X -50.925,Y -35.719,Z -106.683,A -90.000,B 90.000,C 0.000} C_DIS
LIN {X -144.015,Y -35.719,Z -106.683,A -90.000,B 90.000,C 0.000} C_DIS
LIN {X -144.015,Y -35.719,Z -99.134,A -90.000,B 90.000,C 0.000} C_DIS
LIN {X -55.733,Y -35.719,Z -99.134,A -90.000,B 90.000,C 0.000} C_DIS
LIN {X -56.473,Y -35.719,Z -97.666,A -90.000,B 90.000,C 0.000} C_DIS
LIN {X -57.168,Y -35.719,Z -96.176,A -90.000,B 90.000,C 0.000} C_DIS
LIN {X -57.815,Y -35.719,Z -94.665,A -90.000,B 90.000,C 0.000} C_DIS
LIN {X -58.416,Y -35.719,Z -93.134,A -90.000,B 90.000,C 0.000} C_DIS
LIN {X -58.969,Y -35.719,Z -91.586,A -90.000,B 90.000,C 0.000} C_DIS
LIN {X -144.015,Y -35.719,Z -91.586,A -90.000,B 90.000,C 0.000} C_DIS
LIN {X -144.015,Y -35.719,Z -84.037,A -90.000,B 90.000,C 0.000} C_DIS
LIN {X -60.926,Y -35.719,Z -84.037,A -90.000,B 90.000,C 0.000} C_DIS
LIN {X -61.151,Y -35.719,Z -82.705,A -90.000,B 90.000,C 0.000} C_DIS
LIN {X -61.342,Y -35.719,Z -81.367,A -90.000,B 90.000,C 0.000} C_DIS
LIN {X -61.506,Y -35.719,Z -80.154,A -90.000,B 90.000,C 0.000} C_DIS
LIN {X -61.618,Y -35.719,Z -78.935,A -90.000,B 90.000,C 0.000} C_DIS
LIN {X -61.678,Y -35.719,Z -77.712,A -90.000,B 90.000,C 0.000} C_DIS
LIN {X -61.686,Y -35.719,Z -76.488,A -90.000,B 90.000,C 0.000} C_DIS
LIN {X -144.015,Y -35.719,Z -76.488,A -90.000,B 90.000,C 0.000} C_DIS
LIN {X -144.015,Y -35.719,Z -68.939,A -90.000,B 90.000,C 0.000} C_DIS
LIN {X -60.564,Y -35.719,Z -68.939,A -90.000,B 90.000,C 0.000} C_DIS
LIN {X -60.535,Y -35.719,Z -68.840,A -90.000,B 90.000,C 0.000} C_DIS
LIN {X -60.278,Y -35.719,Z -67.814,A -90.000,B 90.000,C 0.000} C_DIS
LIN {X -59.954,Y -35.719,Z -66.806,A -90.000,B 90.000,C 0.000} C_DIS
LIN {X -59.566,Y -35.719,Z -65.822,A -90.000,B 90.000,C 0.000} C_DIS
LIN {X -59.114,Y -35.719,Z -64.865,A -90.000,B 90.000,C 0.000} C_DIS
LIN {X -58.601,Y -35.719,Z -63.940,A -90.000,B 90.000,C 0.000} C_DIS
LIN {X -58.029,Y -35.719,Z -63.050,A -90.000,B 90.000,C 0.000} C_DIS
LIN {X -57.400,Y -35.719,Z -62.199,A -90.000,B 90.000,C 0.000} C_DIS
LIN {X -56.718,Y -35.719,Z -61.390,A -90.000,B 90.000,C 0.000} C_DIS
LIN {X -144.015,Y -35.719,Z -61.390,A -90.000,B 90.000,C 0.000} C_DIS
LIN {X -144.015,Y -35.719,Z -53.842,A -90.000,B 90.000,C 0.000} C_DIS
LIN {X -22.734,Y -35.719,Z -53.842,A -90.000,B 90.000,C 0.000} C_DIS
LIN {X -21.770,Y -35.719,Z -53.355,A -90.000,B 90.000,C 0.000} C_DIS
LIN {X -20.780,Y -35.719,Z -52.924,A -90.000,B 90.000,C 0.000} C_DIS
LIN {X -19.766,Y -35.719,Z -52.552,A -90.000,B 90.000,C 0.000} C_DIS
LIN {X -18.732,Y -35.719,Z -52.238,A -90.000,B 90.000,C 0.000} C_DIS
LIN {X -17.682,Y -35.719,Z -51.986,A -90.000,B 90.000,C 0.000} C_DIS
LIN {X -16.258,Y -35.719,Z -51.827,A -90.000,B 90.000,C 0.000} C_DIS
LIN {X -14.829,Y -35.719,Z -51.728,A -90.000,B 90.000,C 0.000} C_DIS
LIN {X -13.396,Y -35.719,Z -51.687,A -90.000,B 90.000,C 0.000} C_DIS
LIN {X -11.964,Y -35.719,Z -51.704,A -90.000,B 90.000,C 0.000} C_DIS
LIN {X -10.533,Y -35.719,Z -51.780,A -90.000,B 90.000,C 0.000} C_DIS
LIN {X 21.947,Y -35.719,Z -46.293,A -90.000,B 90.000,C 0.000} C_DIS
LIN {X -144.015,Y -35.719,Z -46.293,A -90.000,B 90.000,C 0.000} C_DIS
LIN {X -144.015,Y -35.719,Z -38.744,A -90.000,B 90.000,C 0.000} C_DIS
LIN {X 30.794,Y -35.719,Z -38.744,A -90.000,B 90.000,C 0.000} C_DIS
LIN {X 31.739,Y -35.719,Z -38.446,A -90.000,B 90.000,C 0.000} C_DIS
LIN {X 32.698,Y -35.719,Z -38.202,A -90.000,B 90.000,C 0.000} C_DIS
LIN {X 33.670,Y -35.719,Z -38.013,A -90.000,B 90.000,C 0.000} C_DIS
LIN {X 34.652,Y -35.719,Z -37.880,A -90.000,B 90.000,C 0.000} C_DIS
LIN {X 35.639,Y -35.719,Z -37.802,A -90.000,B 90.000,C 0.000} C_DIS
LIN {X 37.430,Y -35.719,Z -37.937,A -90.000,B 90.000,C 0.000} C_DIS
LIN {X 39.219,Y -35.719,Z -38.105,A -90.000,B 90.000,C 0.000} C_DIS
LIN {X 41.004,Y -35.719,Z -38.305,A -90.000,B 90.000,C 0.000} C_DIS
LIN {X 42.239,Y -35.719,Z -37.979,A -90.000,B 90.000,C 0.000} C_DIS
LIN {X 43.488,Y -35.719,Z -37.713,A -90.000,B 90.000,C 0.000} C_DIS
LIN {X 44.749,Y -35.719,Z -37.510,A -90.000,B 90.000,C 0.000} C_DIS
LIN {X 46.018,Y -35.719,Z -37.369,A -90.000,B 90.000,C 0.000} C_DIS
LIN {X 47.293,Y -35.719,Z -37.290,A -90.000,B 90.000,C 0.000} C_DIS
LIN {X 48.570,Y -35.719,Z -37.275,A -90.000,B 90.000,C 0.000} C_DIS
LIN {X 49.846,Y -35.719,Z -37.322,A -90.000,B 90.000,C 0.000} C_DIS
LIN {X 51.155,Y -35.719,Z -37.590,A -90.000,B 90.000,C 0.000} C_DIS
LIN {X 52.451,Y -35.719,Z -37.917,A -90.000,B 90.000,C 0.000} C_DIS
LIN {X 53.731,Y -35.719,Z -38.302,A -90.000,B 90.000,C 0.000} C_DIS
LIN {X 54.992,Y -35.719,Z -38.744,A -90.000,B 90.000,C 0.000} C_DIS
LIN {X 87.858,Y -35.719,Z -38.744,A -90.000,B 90.000,C 0.000} C_DIS
LIN {X 87.334,Y -35.719,Z -39.544,A -90.000,B 90.000,C 0.000} C_DIS
LIN {X 86.855,Y -35.719,Z -40.373,A -90.000,B 90.000,C 0.000} C_DIS
LIN {X 86.425,Y -35.719,Z -41.227,A -90.000,B 90.000,C 0.000} C_DIS
LIN {X 86.042,Y -35.719,Z -42.104,A -90.000,B 90.000,C 0.000} C_DIS
LIN {X 85.710,Y -35.719,Z -43.001,A -90.000,B 90.000,C 0.000} C_DIS
LIN {X 85.429,Y -35.719,Z -43.916,A -90.000,B 90.000,C 0.000} C_DIS
LIN {X 85.201,Y -35.719,Z -44.845,A -90.000,B 90.000,C 0.000} C_DIS
LIN {X 85.118,Y -35.719,Z -45.325,A -90.000,B 90.000,C 0.000} C_DIS
LIN {X 85.057,Y -35.719,Z -45.808,A -90.000,B 90.000,C 0.000} C_DIS
LIN {X 85.018,Y -35.719,Z -46.293,A -90.000,B 90.000,C 0.000} C_DIS
LIN {X 66.046,Y -35.719,Z -46.293,A -90.000,B 90.000,C 0.000} C_DIS
LIN {X 67.465,Y -35.719,Z -47.652,A -90.000,B 90.000,C 0.000} C_DIS
LIN {X 68.908,Y -35.719,Z -48.986,A -90.000,B 90.000,C 0.000} C_DIS
LIN {X 70.373,Y -35.719,Z -50.296,A -90.000,B 90.000,C 0.000} C_DIS
LIN {X 71.860,Y -35.719,Z -51.580,A -90.000,B 90.000,C 0.000} C_DIS
LIN {X 72.759,Y -35.719,Z -52.305,A -90.000,B 90.000,C 0.000} C_DIS
LIN {X 73.633,Y -35.719,Z -53.059,A -90.000,B 90.000,C 0.000} C_DIS
LIN {X 74.482,Y -35.719,Z -53.842,A -90.000,B 90.000,C 0.000} C_DIS
LIN {X 79.082,Y -35.719,Z -53.842,A -90.000,B 90.000,C 0.000} C_DIS
LIN {X 79.386,Y -35.719,Z -53.483,A -90.000,B 90.000,C 0.000} C_DIS
LIN {X 85.001,Y -35.719,Z -46.864,A -90.000,B 90.000,C 0.000} C_DIS
LIN {X 85.024,Y -35.719,Z -46.187,A -90.000,B 90.000,C 0.000} C_DIS
LIN {X 85.091,Y -35.719,Z -45.513,A -90.000,B 90.000,C 0.000} C_DIS
LIN {X 85.201,Y -35.719,Z -44.845,A -90.000,B 90.000,C 0.000} C_DIS
LIN {X 85.451,Y -35.719,Z -43.840,A -90.000,B 90.000,C 0.000} C_DIS
LIN {X 85.762,Y -35.719,Z -42.852,A -90.000,B 90.000,C 0.000} C_DIS
LIN {X 86.133,Y -35.719,Z -41.885,A -90.000,B 90.000,C 0.000} C_DIS
LIN {X 86.562,Y -35.719,Z -40.943,A -90.000,B 90.000,C 0.000} C_DIS
LIN {X 87.048,Y -35.719,Z -40.028,A -90.000,B 90.000,C 0.000} C_DIS
LIN {X 87.588,Y -35.719,Z -39.144,A -90.000,B 90.000,C 0.000} C_DIS
LIN {X 88.182,Y -35.719,Z -38.296,A -90.000,B 90.000,C 0.000} C_DIS
LIN {X 88.826,Y -35.719,Z -37.485,A -90.000,B 90.000,C 0.000} C_DIS
LIN {X 89.518,Y -35.719,Z -36.714,A -90.000,B 90.000,C 0.000} C_DIS
LIN {X 90.256,Y -35.719,Z -35.988,A -90.000,B 90.000,C 0.000} C_DIS
LIN {X 91.037,Y -35.719,Z -35.308,A -90.000,B 90.000,C 0.000} C_DIS
LIN {X 91.858,Y -35.719,Z -34.677,A -90.000,B 90.000,C 0.000} C_DIS
LIN {X 92.716,Y -35.719,Z -34.096,A -90.000,B 90.000,C 0.000} C_DIS
LIN {X 94.550,Y -35.719,Z -33.081,A -90.000,B 90.000,C 0.000} C_DIS
LIN {X 96.409,Y -35.719,Z -32.114,A -90.000,B 90.000,C 0.000} C_DIS
LIN {X 98.293,Y -35.719,Z -31.195,A -90.000,B 90.000,C 0.000} C_DIS
LIN {X -144.015,Y -35.719,Z -31.195,A -90.000,B 90.000,C 0.000} C_DIS
LIN {X -144.015,Y -35.719,Z -23.646,A -90.000,B 90.000,C 0.000} C_DIS
LIN {X 144.015,Y -35.719,Z -23.646,A -90.000,B 90.000,C 0.000} C_DIS
LIN {X 144.015,Y -35.719,Z -16.098,A -90.000,B 90.000,C 0.000} C_DIS
LIN {X -144.015,Y -35.719,Z -16.098,A -90.000,B 90.000,C 0.000} C_DIS
LIN {X -144.015,Y -35.719,Z -8.549,A -90.000,B 90.000,C 0.000} C_DIS
LIN {X 144.015,Y -35.719,Z -8.549,A -90.000,B 90.000,C 0.000} C_DIS
LIN {X 144.015,Y -35.719,Z -1.000,A -90.000,B 90.000,C 0.000} C_DIS
LIN {X -144.015,Y -35.719,Z -1.000,A -90.000,B 90.000,C 0.000} C_DIS
LIN {X 102.939,Y -35.719,Z -29.179,A -90.000,B 90.000,C 0.000} C_DIS
LIN {X 103.563,Y -35.719,Z -28.934,A -90.000,B 90.000,C 0.000} C_DIS
LIN {X 104.190,Y -35.719,Z -28.694,A -90.000,B 90.000,C 0.000} C_DIS
LIN {X 105.127,Y -35.719,Z -28.308,A -90.000,B 90.000,C 0.000} C_DIS
LIN {X 106.088,Y -35.719,Z -27.985,A -90.000,B 90.000,C 0.000} C_DIS
LIN {X 107.068,Y -35.719,Z -27.726,A -90.000,B 90.000,C 0.000} C_DIS
LIN {X 108.063,Y -35.719,Z -27.533,A -90.000,B 90.000,C 0.000} C_DIS
LIN {X 109.069,Y -35.719,Z -27.406,A -90.000,B 90.000,C 0.000} C_DIS
LIN {X 110.081,Y -35.719,Z -27.346,A -90.000,B 90.000,C 0.000} C_DIS
LIN {X 111.095,Y -35.719,Z -27.353,A -90.000,B 90.000,C 0.000} C_DIS
LIN {X 112.106,Y -35.719,Z -27.427,A -90.000,B 90.000,C 0.000} C_DIS
LIN {X 113.109,Y -35.719,Z -27.568,A -90.000,B 90.000,C 0.000} C_DIS
LIN {X 114.102,Y -35.719,Z -27.775,A -90.000,B 90.000,C 0.000} C_DIS
LIN {X 115.078,Y -35.719,Z -28.047,A -90.000,B 90.000,C 0.000} C_DIS
LIN {X 116.034,Y -35.719,Z -28.383,A -90.000,B 90.000,C 0.000} C_DIS
LIN {X 116.966,Y -35.719,Z -28.782,A -90.000,B 90.000,C 0.000} C_DIS
LIN {X 117.870,Y -35.719,Z -29.242,A -90.000,B 90.000,C 0.000} C_DIS
LIN {X 118.741,Y -35.719,Z -29.761,A -90.000,B 90.000,C 0.000} C_DIS
LIN {X 119.576,Y -35.719,Z -30.335,A -90.000,B 90.000,C 0.000} C_DIS
LIN {X 119.743,Y -35.719,Z -30.461,A -90.000,B 90.000,C 0.000} C_DIS
LIN {X 120.184,Y -35.719,Z -30.821,A -90.000,B 90.000,C 0.000} C_DIS
LIN {X 120.612,Y -35.719,Z -31.195,A -90.000,B 90.000,C 0.000} C_DIS
LIN {X 144.015,Y -35.719,Z -31.195,A -90.000,B 90.000,C 0.000} C_DIS
LIN {X 144.015,Y -35.719,Z -38.744,A -90.000,B 90.000,C 0.000} C_DIS
LIN {X 124.956,Y -35.719,Z -38.744,A -90.000,B 90.000,C 0.000} C_DIS
LIN {X 125.148,Y -35.719,Z -39.640,A -90.000,B 90.000,C 0.000} C_DIS
LIN {X 125.291,Y -35.719,Z -40.545,A -90.000,B 90.000,C 0.000} C_DIS
LIN {X 125.384,Y -35.719,Z -41.456,A -90.000,B 90.000,C 0.000} C_DIS
LIN {X 125.427,Y -35.719,Z -42.371,A -90.000,B 90.000,C 0.000} C_DIS
LIN {X 125.420,Y -35.719,Z -43.288,A -90.000,B 90.000,C 0.000} C_DIS
LIN {X 125.363,Y -35.719,Z -44.202,A -90.000,B 90.000,C 0.000} C_DIS
LIN {X 125.205,Y -35.719,Z -45.251,A -90.000,B 90.000,C 0.000} C_DIS
LIN {X 125.008,Y -35.719,Z -46.293,A -90.000,B 90.000,C 0.000} C_DIS
LIN {X 144.015,Y -35.719,Z -46.293,A -90.000,B 90.000,C 0.000} C_DIS
LIN {X 144.015,Y -35.719,Z -53.842,A -90.000,B 90.000,C 0.000} C_DIS
LIN {X 122.267,Y -35.719,Z -53.842,A -90.000,B 90.000,C 0.000} C_DIS
LIN {X 121.511,Y -35.719,Z -55.301,A -90.000,B 90.000,C 0.000} C_DIS
LIN {X 120.810,Y -35.719,Z -56.787,A -90.000,B 90.000,C 0.000} C_DIS
LIN {X 120.167,Y -35.719,Z -58.299,A -90.000,B 90.000,C 0.000} C_DIS
LIN {X 119.581,Y -35.719,Z -59.834,A -90.000,B 90.000,C 0.000} C_DIS
LIN {X 119.054,Y -35.719,Z -61.390,A -90.000,B 90.000,C 0.000} C_DIS
LIN {X 144.015,Y -35.719,Z -61.390,A -90.000,B 90.000,C 0.000} C_DIS
LIN {X 144.015,Y -35.719,Z -68.939,A -90.000,B 90.000,C 0.000} C_DIS
LIN {X 116.899,Y -35.719,Z -68.939,A -90.000,B 90.000,C 0.000} C_DIS
LIN {X 116.228,Y -35.719,Z -70.853,A -90.000,B 90.000,C 0.000} C_DIS
LIN {X 115.511,Y -35.719,Z -72.750,A -90.000,B 90.000,C 0.000} C_DIS
LIN {X 114.747,Y -35.719,Z -74.629,A -90.000,B 90.000,C 0.000} C_DIS
LIN {X 113.936,Y -35.719,Z -76.488,A -90.000,B 90.000,C 0.000} C_DIS
LIN {X 144.015,Y -35.719,Z -76.488,A -90.000,B 90.000,C 0.000} C_DIS
LIN {X 144.015,Y -35.719,Z -84.037,A -90.000,B 90.000,C 0.000} C_DIS
LIN {X 110.056,Y -35.719,Z -84.037,A -90.000,B 90.000,C 0.000} C_DIS
LIN {X 109.198,Y -35.719,Z -85.479,A -90.000,B 90.000,C 0.000} C_DIS
LIN {X 108.312,Y -35.719,Z -86.903,A -90.000,B 90.000,C 0.000} C_DIS
LIN {X 107.396,Y -35.719,Z -88.308,A -90.000,B 90.000,C 0.000} C_DIS
LIN {X 106.452,Y -35.719,Z -89.695,A -90.000,B 90.000,C 0.000} C_DIS
LIN {X 106.402,Y -35.719,Z -90.413,A -90.000,B 90.000,C 0.000} C_DIS
LIN {X 106.339,Y -35.719,Z -91.130,A -90.000,B 90.000,C 0.000} C_DIS
LIN {X 106.338,Y -35.719,Z -91.586,A -90.000,B 90.000,C 0.000} C_DIS
LIN {X 144.015,Y -35.719,Z -91.586,A -90.000,B 90.000,C 0.000} C_DIS
LIN {X 144.015,Y -35.719,Z -99.134,A -90.000,B 90.000,C 0.000} C_DIS
LIN {X 105.264,Y -35.719,Z -99.134,A -90.000,B 90.000,C 0.000} C_DIS
LIN {X 105.119,Y -35.719,Z -99.637,A -90.000,B 90.000,C 0.000} C_DIS
LIN {X 104.800,Y -35.719,Z -100.509,A -90.000,B 90.000,C 0.000} C_DIS
LIN {X 104.519,Y -35.719,Z -101.395,A -90.000,B 90.000,C 0.000} C_DIS
LIN {X 104.277,Y -35.719,Z -102.292,A -90.000,B 90.000,C 0.000} C_DIS
LIN {X 104.075,Y -35.719,Z -103.199,A -90.000,B 90.000,C 0.000} C_DIS
LIN {X 104.047,Y -35.719,Z -103.340,A -90.000,B 90.000,C 0.000} C_DIS
LIN {X 103.980,Y -35.719,Z -103.468,A -90.000,B 90.000,C 0.000} C_DIS
LIN {X 103.824,Y -35.719,Z -103.821,A -90.000,B 90.000,C 0.000} C_DIS
LIN {X 103.716,Y -35.719,Z -104.192,A -90.000,B 90.000,C 0.000} C_DIS
LIN {X 103.657,Y -35.719,Z -104.574,A -90.000,B 90.000,C 0.000} C_DIS
LIN {X 103.650,Y -35.719,Z -104.960,A -90.000,B 90.000,C 0.000} C_DIS
LIN {X 103.694,Y -35.719,Z -105.344,A -90.000,B 90.000,C 0.000} C_DIS
LIN {X 103.788,Y -35.719,Z -105.718,A -90.000,B 90.000,C 0.000} C_DIS
LIN {X 103.864,Y -35.719,Z -106.683,A -90.000,B 90.000,C 0.000} C_DIS
LIN {X 144.015,Y -35.719,Z -106.683,A -90.000,B 90.000,C 0.000} C_DIS
LIN {X 144.015,Y -35.719,Z -114.232,A -90.000,B 90.000,C 0.000} C_DIS
LIN {X 104.169,Y -35.719,Z -114.232,A -90.000,B 90.000,C 0.000} C_DIS
LIN {X 104.171,Y -35.719,Z -115.213,A -90.000,B 90.000,C 0.000} C_DIS
LIN {X 104.164,Y -35.719,Z -116.193,A -90.000,B 90.000,C 0.000} C_DIS
LIN {X 104.228,Y -35.719,Z -118.055,A -90.000,B 90.000,C 0.000} C_DIS
LIN {X 104.266,Y -35.719,Z -119.918,A -90.000,B 90.000,C 0.000} C_DIS
LIN {X 104.278,Y -35.719,Z -121.781,A -90.000,B 90.000,C 0.000} C_DIS
LIN {X 144.015,Y -35.719,Z -121.781,A -90.000,B 90.000,C 0.000} C_DIS
LIN {X 144.015,Y -35.719,Z -129.329,A -90.000,B 90.000,C 0.000} C_DIS
LIN {X 104.053,Y -35.719,Z -129.329,A -90.000,B 90.000,C 0.000} C_DIS
LIN {X 103.914,Y -35.719,Z -131.422,A -90.000,B 90.000,C 0.000} C_DIS
LIN {X 103.741,Y -35.719,Z -133.512,A -90.000,B 90.000,C 0.000} C_DIS
LIN {X 103.536,Y -35.719,Z -135.599,A -90.000,B 90.000,C 0.000} C_DIS
LIN {X 103.466,Y -35.719,Z -136.878,A -90.000,B 90.000,C 0.000} C_DIS
LIN {X 144.015,Y -35.719,Z -136.878,A -90.000,B 90.000,C 0.000} C_DIS
LIN {X 144.015,Y -35.719,Z -144.427,A -90.000,B 90.000,C 0.000} C_DIS
LIN {X 102.837,Y -35.719,Z -144.427,A -90.000,B 90.000,C 0.000} C_DIS
LIN {X 102.544,Y -35.719,Z -146.949,A -90.000,B 90.000,C 0.000} C_DIS
LIN {X 102.210,Y -35.719,Z -149.465,A -90.000,B 90.000,C 0.000} C_DIS
LIN {X 101.835,Y -35.719,Z -151.976,A -90.000,B 90.000,C 0.000} C_DIS
LIN {X 144.015,Y -35.719,Z -151.976,A -90.000,B 90.000,C 0.000} C_DIS
LIN {X 144.015,Y -35.719,Z -159.525,A -90.000,B 90.000,C 0.000} C_DIS
LIN {X 100.431,Y -35.719,Z -159.525,A -90.000,B 90.000,C 0.000} C_DIS
LIN {X 99.835,Y -35.719,Z -162.048,A -90.000,B 90.000,C 0.000} C_DIS
LIN {X 99.212,Y -35.719,Z -164.564,A -90.000,B 90.000,C 0.000} C_DIS
LIN {X 98.561,Y -35.719,Z -167.073,A -90.000,B 90.000,C 0.000} C_DIS
LIN {X 144.015,Y -35.719,Z -167.073,A -90.000,B 90.000,C 0.000} C_DIS
LIN {X 144.015,Y -35.719,Z -174.622,A -90.000,B 90.000,C 0.000} C_DIS
LIN {X 96.429,Y -35.719,Z -174.622,A -90.000,B 90.000,C 0.000} C_DIS
LIN {X 95.638,Y -35.719,Z -177.203,A -90.000,B 90.000,C 0.000} C_DIS
LIN {X 94.819,Y -35.719,Z -179.776,A -90.000,B 90.000,C 0.000} C_DIS
LIN {X 94.054,Y -35.719,Z -182.171,A -90.000,B 90.000,C 0.000} C_DIS
LIN {X 144.015,Y -35.719,Z -182.171,A -90.000,B 90.000,C 0.000} C_DIS
LIN {X 144.015,Y -35.719,Z -189.720,A -90.000,B 90.000,C 0.000} C_DIS
LIN {X 91.645,Y -35.719,Z -189.720,A -90.000,B 90.000,C 0.000} C_DIS
LIN {X 90.574,Y -35.719,Z -193.075,A -90.000,B 90.000,C 0.000} C_DIS
LIN {X 89.891,Y -35.719,Z -195.174,A -90.000,B 90.000,C 0.000} C_DIS
LIN {X 89.197,Y -35.719,Z -197.269,A -90.000,B 90.000,C 0.000} C_DIS
LIN {X 144.015,Y -35.719,Z -197.269,A -90.000,B 90.000,C 0.000} C_DIS
LIN {X 144.015,Y -35.719,Z -204.817,A -90.000,B 90.000,C 0.000} C_DIS
LIN {X 86.584,Y -35.719,Z -204.817,A -90.000,B 90.000,C 0.000} C_DIS
LIN {X 85.209,Y -35.719,Z -208.599,A -90.000,B 90.000,C 0.000} C_DIS
LIN {X 83.794,Y -35.719,Z -212.366,A -90.000,B 90.000,C 0.000} C_DIS
LIN {X 144.015,Y -35.719,Z -212.366,A -90.000,B 90.000,C 0.000} C_DIS
LIN {X 144.015,Y -35.719,Z -219.915,A -90.000,B 90.000,C 0.000} C_DIS
LIN {X 80.823,Y -35.719,Z -219.915,A -90.000,B 90.000,C 0.000} C_DIS
LIN {X 80.067,Y -35.719,Z -221.764,A -90.000,B 90.000,C 0.000} C_DIS
LIN {X 78.838,Y -35.719,Z -224.611,A -90.000,B 90.000,C 0.000} C_DIS
LIN {X 77.622,Y -35.719,Z -227.464,A -90.000,B 90.000,C 0.000} C_DIS
LIN {X 144.015,Y -35.719,Z -227.464,A -90.000,B 90.000,C 0.000} C_DIS
LIN {X 144.015,Y -35.719,Z -235.012,A -90.000,B 90.000,C 0.000} C_DIS
LIN {X 74.469,Y -35.719,Z -235.012,A -90.000,B 90.000,C 0.000} C_DIS
LIN {X 72.930,Y -35.719,Z -238.782,A -90.000,B 90.000,C 0.000} C_DIS
LIN {X 71.411,Y -35.719,Z -242.561,A -90.000,B 90.000,C 0.000} C_DIS
LIN {X 144.015,Y -35.719,Z -242.561,A -90.000,B 90.000,C 0.000} C_DIS
LIN {X 96.155,Y -35.719,Z -175.529,A -90.000,B 90.000,C 0.000} C_DIS
LIN {X 97.152,Y -35.719,Z -172.168,A -90.000,B 90.000,C 0.000} C_DIS
LIN {X 98.099,Y -35.719,Z -168.792,A -90.000,B 90.000,C 0.000} C_DIS
LIN {X 98.998,Y -35.719,Z -165.403,A -90.000,B 90.000,C 0.000} C_DIS
LIN {X 99.846,Y -35.719,Z -162.001,A -90.000,B 90.000,C 0.000} C_DIS
LIN {X 100.645,Y -35.719,Z -158.587,A -90.000,B 90.000,C 0.000} C_DIS
LIN {X 101.194,Y -35.719,Z -155.741,A -90.000,B 90.000,C 0.000} C_DIS
LIN {X 101.689,Y -35.719,Z -152.884,A -90.000,B 90.000,C 0.000} C_DIS
LIN {X 102.131,Y -35.719,Z -150.020,A -90.000,B 90.000,C 0.000} C_DIS
LIN {X 102.519,Y -35.719,Z -147.147,A -90.000,B 90.000,C 0.000} C_DIS
LIN {X 102.854,Y -35.719,Z -144.268,A -90.000,B 90.000,C 0.000} C_DIS
LIN {X 103.135,Y -35.719,Z -141.382,A -90.000,B 90.000,C 0.000} C_DIS
LIN {X 103.362,Y -35.719,Z -138.493,A -90.000,B 90.000,C 0.000} C_DIS
LIN {X 103.536,Y -35.719,Z -135.599,A -90.000,B 90.000,C 0.000} C_DIS
LIN {X 103.801,Y -35.719,Z -132.835,A -90.000,B 90.000,C 0.000} C_DIS
LIN {X 104.009,Y -35.719,Z -130.067,A -90.000,B 90.000,C 0.000} C_DIS
LIN {X 104.157,Y -35.719,Z -127.295,A -90.000,B 90.000,C 0.000} C_DIS
LIN {X 104.247,Y -35.719,Z -124.520,A -90.000,B 90.000,C 0.000} C_DIS
LIN {X 104.278,Y -35.719,Z -121.744,A -90.000,B 90.000,C 0.000} C_DIS
LIN {X 104.251,Y -35.719,Z -118.968,A -90.000,B 90.000,C 0.000} C_DIS
LIN {X 104.164,Y -35.719,Z -116.193,A -90.000,B 90.000,C 0.000} C_DIS
LIN {X 104.167,Y -35.719,Z -114.096,A -90.000,B 90.000,C 0.000} C_DIS
LIN {X 104.131,Y -35.719,Z -111.999,A -90.000,B 90.000,C 0.000} C_DIS
LIN {X 104.056,Y -35.719,Z -109.903,A -90.000,B 90.000,C 0.000} C_DIS
LIN {X 103.942,Y -35.719,Z -107.809,A -90.000,B 90.000,C 0.000} C_DIS
LIN {X 103.788,Y -35.719,Z -105.718,A -90.000,B 90.000,C 0.000} C_DIS
LIN {X 103.694,Y -35.719,Z -105.343,A -90.000,B 90.000,C 0.000} C_DIS
LIN {X 103.650,Y -35.719,Z -104.960,A -90.000,B 90.000,C 0.000} C_DIS
LIN {X 103.658,Y -35.719,Z -104.574,A -90.000,B 90.000,C 0.000} C_DIS
LIN {X 103.716,Y -35.719,Z -104.192,A -90.000,B 90.000,C 0.000} C_DIS
LIN {X 103.824,Y -35.719,Z -103.821,A -90.000,B 90.000,C 0.000} C_DIS
LIN {X 103.980,Y -35.719,Z -103.468,A -90.000,B 90.000,C 0.000} C_DIS
LIN {X 104.047,Y -35.719,Z -103.340,A -90.000,B 90.000,C 0.000} C_DIS
LIN {X 104.075,Y -35.719,Z -103.199,A -90.000,B 90.000,C 0.000} C_DIS
LIN {X 104.277,Y -35.719,Z -102.292,A -90.000,B 90.000,C 0.000} C_DIS
LIN {X 104.518,Y -35.719,Z -101.395,A -90.000,B 90.000,C 0.000} C_DIS
LIN {X 104.799,Y -35.719,Z -100.509,A -90.000,B 90.000,C 0.000} C_DIS
LIN {X 105.119,Y -35.719,Z -99.637,A -90.000,B 90.000,C 0.000} C_DIS
LIN {X 105.447,Y -35.719,Z -98.449,A -90.000,B 90.000,C 0.000} C_DIS
LIN {X 105.724,Y -35.719,Z -97.249,A -90.000,B 90.000,C 0.000} C_DIS
LIN {X 105.951,Y -35.719,Z -96.038,A -90.000,B 90.000,C 0.000} C_DIS
LIN {X 106.126,Y -35.719,Z -94.818,A -90.000,B 90.000,C 0.000} C_DIS
LIN {X 106.249,Y -35.719,Z -93.592,A -90.000,B 90.000,C 0.000} C_DIS
LIN {X 106.320,Y -35.719,Z -92.362,A -90.000,B 90.000,C 0.000} C_DIS
LIN {X 106.339,Y -35.719,Z -91.130,A -90.000,B 90.000,C 0.000} C_DIS
LIN {X 106.402,Y -35.719,Z -90.413,A -90.000,B 90.000,C 0.000} C_DIS
LIN {X 106.452,Y -35.719,Z -89.695,A -90.000,B 90.000,C 0.000} C_DIS
LIN {X 107.788,Y -35.719,Z -87.715,A -90.000,B 90.000,C 0.000} C_DIS
LIN {X 109.065,Y -35.719,Z -85.696,A -90.000,B 90.000,C 0.000} C_DIS
LIN {X 110.284,Y -35.719,Z -83.642,A -90.000,B 90.000,C 0.000} C_DIS
LIN {X 111.442,Y -35.719,Z -81.553,A -90.000,B 90.000,C 0.000} C_DIS
LIN {X 112.540,Y -35.719,Z -79.431,A -90.000,B 90.000,C 0.000} C_DIS
LIN {X 113.575,Y -35.719,Z -77.278,A -90.000,B 90.000,C 0.000} C_DIS
LIN {X 114.548,Y -35.719,Z -75.096,A -90.000,B 90.000,C 0.000} C_DIS
LIN {X 115.456,Y -35.719,Z -72.887,A -90.000,B 90.000,C 0.000} C_DIS
LIN {X 116.300,Y -35.719,Z -70.653,A -90.000,B 90.000,C 0.000} C_DIS
LIN {X 117.080,Y -35.719,Z -68.394,A -90.000,B 90.000,C 0.000} C_DIS
LIN {X 117.793,Y -35.719,Z -66.115,A -90.000,B 90.000,C 0.000} C_DIS
LIN {X 118.440,Y -35.719,Z -63.815,A -90.000,B 90.000,C 0.000} C_DIS
LIN {X 119.020,Y -35.719,Z -61.498,A -90.000,B 90.000,C 0.000} C_DIS
LIN {X 119.501,Y -35.719,Z -60.058,A -90.000,B 90.000,C 0.000} C_DIS
LIN {X 120.032,Y -35.719,Z -58.637,A -90.000,B 90.000,C 0.000} C_DIS
LIN {X 120.613,Y -35.719,Z -57.234,A -90.000,B 90.000,C 0.000} C_DIS
LIN {X 121.242,Y -35.719,Z -55.853,A -90.000,B 90.000,C 0.000} C_DIS
LIN {X 121.920,Y -35.719,Z -54.495,A -90.000,B 90.000,C 0.000} C_DIS
LIN {X 122.644,Y -35.719,Z -53.161,A -90.000,B 90.000,C 0.000} C_DIS
LIN {X 123.210,Y -35.719,Z -51.943,A -90.000,B 90.000,C 0.000} C_DIS
LIN {X 123.718,Y -35.719,Z -50.699,A -90.000,B 90.000,C 0.000} C_DIS
LIN {X 124.168,Y -35.719,Z -49.433,A -90.000,B 90.000,C 0.000} C_DIS
LIN {X 124.558,Y -35.719,Z -48.148,A -90.000,B 90.000,C 0.000} C_DIS
LIN {X 124.887,Y -35.719,Z -46.845,A -90.000,B 90.000,C 0.000} C_DIS
LIN {X 125.156,Y -35.719,Z -45.529,A -90.000,B 90.000,C 0.000} C_DIS
LIN {X 125.363,Y -35.719,Z -44.202,A -90.000,B 90.000,C 0.000} C_DIS
LIN {X 125.424,Y -35.719,Z -43.147,A -90.000,B 90.000,C 0.000} C_DIS
LIN {X 125.419,Y -35.719,Z -42.091,A -90.000,B 90.000,C 0.000} C_DIS
LIN {X 125.347,Y -35.719,Z -41.037,A -90.000,B 90.000,C 0.000} C_DIS
LIN {X 125.209,Y -35.719,Z -39.989,A -90.000,B 90.000,C 0.000} C_DIS
LIN {X 125.005,Y -35.719,Z -38.953,A -90.000,B 90.000,C 0.000} C_DIS
LIN {X 124.737,Y -35.719,Z -37.931,A -90.000,B 90.000,C 0.000} C_DIS
LIN {X 124.404,Y -35.719,Z -36.928,A -90.000,B 90.000,C 0.000} C_DIS
LIN {X 124.009,Y -35.719,Z -35.948,A -90.000,B 90.000,C 0.000} C_DIS
LIN {X 123.553,Y -35.719,Z -34.995,A -90.000,B 90.000,C 0.000} C_DIS
LIN {X 123.038,Y -35.719,Z -34.073,A -90.000,B 90.000,C 0.000} C_DIS
LIN {X 122.466,Y -35.719,Z -33.185,A -90.000,B 90.000,C 0.000} C_DIS
LIN {X 122.381,Y -35.719,Z -33.078,A -90.000,B 90.000,C 0.000} C_DIS
LIN {X 121.779,Y -35.719,Z -32.368,A -90.000,B 90.000,C 0.000} C_DIS
LIN {X 121.137,Y -35.719,Z -31.694,A -90.000,B 90.000,C 0.000} C_DIS
LIN {X 120.458,Y -35.719,Z -31.057,A -90.000,B 90.000,C 0.000} C_DIS
LIN {X 119.743,Y -35.719,Z -30.461,A -90.000,B 90.000,C 0.000} C_DIS
LIN {X 119.576,Y -35.719,Z -30.335,A -90.000,B 90.000,C 0.000} C_DIS
LIN {X 118.741,Y -35.719,Z -29.760,A -90.000,B 90.000,C 0.000} C_DIS
LIN {X 117.870,Y -35.719,Z -29.241,A -90.000,B 90.000,C 0.000} C_DIS
LIN {X 116.967,Y -35.719,Z -28.782,A -90.000,B 90.000,C 0.000} C_DIS
LIN {X 116.035,Y -35.719,Z -28.383,A -90.000,B 90.000,C 0.000} C_DIS
LIN {X 115.078,Y -35.719,Z -28.046,A -90.000,B 90.000,C 0.000} C_DIS
LIN {X 114.102,Y -35.719,Z -27.774,A -90.000,B 90.000,C 0.000} C_DIS
LIN {X 113.110,Y -35.719,Z -27.567,A -90.000,B 90.000,C 0.000} C_DIS
LIN {X 112.106,Y -35.719,Z -27.426,A -90.000,B 90.000,C 0.000} C_DIS
LIN {X 111.095,Y -35.719,Z -27.352,A -90.000,B 90.000,C 0.000} C_DIS
LIN {X 110.081,Y -35.719,Z -27.345,A -90.000,B 90.000,C 0.000} C_DIS
LIN {X 109.069,Y -35.719,Z -27.405,A -90.000,B 90.000,C 0.000} C_DIS
LIN {X 108.063,Y -35.719,Z -27.532,A -90.000,B 90.000,C 0.000} C_DIS
LIN {X 107.068,Y -35.719,Z -27.725,A -90.000,B 90.000,C 0.000} C_DIS
LIN {X 106.088,Y -35.719,Z -27.984,A -90.000,B 90.000,C 0.000} C_DIS
LIN {X 105.127,Y -35.719,Z -28.307,A -90.000,B 90.000,C 0.000} C_DIS
LIN {X 104.190,Y -35.719,Z -28.694,A -90.000,B 90.000,C 0.000} C_DIS
LIN {X 102.221,Y -35.719,Z -29.468,A -90.000,B 90.000,C 0.000} C_DIS
LIN {X 100.273,Y -35.719,Z -30.294,A -90.000,B 90.000,C 0.000} C_DIS
LIN {X 98.347,Y -35.719,Z -31.170,A -90.000,B 90.000,C 0.000} C_DIS
LIN {X 96.445,Y -35.719,Z -32.096,A -90.000,B 90.000,C 0.000} C_DIS
LIN {X 94.567,Y -35.719,Z -33.072,A -90.000,B 90.000,C 0.000} C_DIS
LIN {X 92.716,Y -35.719,Z -34.096,A -90.000,B 90.000,C 0.000} C_DIS
LIN {X 91.858,Y -35.719,Z -34.676,A -90.000,B 90.000,C 0.000} C_DIS
LIN {X 91.037,Y -35.719,Z -35.307,A -90.000,B 90.000,C 0.000} C_DIS
LIN {X 90.256,Y -35.719,Z -35.987,A -90.000,B 90.000,C 0.000} C_DIS
LIN {X 89.518,Y -35.719,Z -36.714,A -90.000,B 90.000,C 0.000} C_DIS
LIN {X 88.825,Y -35.719,Z -37.484,A -90.000,B 90.000,C 0.000} C_DIS
LIN {X 88.181,Y -35.719,Z -38.295,A -90.000,B 90.000,C 0.000} C_DIS
LIN {X 87.588,Y -35.719,Z -39.144,A -90.000,B 90.000,C 0.000} C_DIS
LIN {X 87.047,Y -35.719,Z -40.027,A -90.000,B 90.000,C 0.000} C_DIS
LIN {X 86.561,Y -35.719,Z -40.942,A -90.000,B 90.000,C 0.000} C_DIS
LIN {X 86.132,Y -35.719,Z -41.885,A -90.000,B 90.000,C 0.000} C_DIS
LIN {X 85.762,Y -35.719,Z -42.852,A -90.000,B 90.000,C 0.000} C_DIS
LIN {X 85.451,Y -35.719,Z -43.840,A -90.000,B 90.000,C 0.000} C_DIS
LIN {X 85.201,Y -35.719,Z -44.845,A -90.000,B 90.000,C 0.000} C_DIS
LIN {X 85.086,Y -35.719,Z -45.557,A -90.000,B 90.000,C 0.000} C_DIS
LIN {X 85.019,Y -35.719,Z -46.275,A -90.000,B 90.000,C 0.000} C_DIS
LIN {X 85.002,Y -35.719,Z -46.996,A -90.000,B 90.000,C 0.000} C_DIS
LIN {X 85.033,Y -35.719,Z -47.716,A -90.000,B 90.000,C 0.000} C_DIS
LIN {X 83.572,Y -35.719,Z -49.063,A -90.000,B 90.000,C 0.000} C_DIS
LIN {X 82.157,Y -35.719,Z -50.458,A -90.000,B 90.000,C 0.000} C_DIS
LIN {X 80.788,Y -35.719,Z -51.900,A -90.000,B 90.000,C 0.000} C_DIS
LIN {X 79.469,Y -35.719,Z -53.386,A -90.000,B 90.000,C 0.000} C_DIS
LIN {X 78.199,Y -35.719,Z -54.915,A -90.000,B 90.000,C 0.000} C_DIS
LIN {X 76.981,Y -35.719,Z -56.485,A -90.000,B 90.000,C 0.000} C_DIS
LIN {X 76.038,Y -35.719,Z -55.422,A -90.000,B 90.000,C 0.000} C_DIS
LIN {X 75.053,Y -35.719,Z -54.399,A -90.000,B 90.000,C 0.000} C_DIS
LIN {X 74.027,Y -35.719,Z -53.416,A -90.000,B 90.000,C 0.000} C_DIS
LIN {X 72.962,Y -35.719,Z -52.476,A -90.000,B 90.000,C 0.000} C_DIS
LIN {X 71.860,Y -35.719,Z -51.580,A -90.000,B 90.000,C 0.000} C_DIS
LIN {X 70.287,Y -35.719,Z -50.220,A -90.000,B 90.000,C 0.000} C_DIS
LIN {X 68.738,Y -35.719,Z -48.832,A -90.000,B 90.000,C 0.000} C_DIS
LIN {X 67.216,Y -35.719,Z -47.417,A -90.000,B 90.000,C 0.000} C_DIS
LIN {X 65.719,Y -35.719,Z -45.973,A -90.000,B 90.000,C 0.000} C_DIS
LIN {X 64.563,Y -35.719,Z -44.880,A -90.000,B 90.000,C 0.000} C_DIS
LIN {X 63.360,Y -35.719,Z -43.837,A -90.000,B 90.000,C 0.000} C_DIS
LIN {X 62.113,Y -35.719,Z -42.849,A -90.000,B 90.000,C 0.000} C_DIS
LIN {X 60.824,Y -35.719,Z -41.915,A -90.000,B 90.000,C 0.000} C_DIS
LIN {X 59.496,Y -35.719,Z -41.038,A -90.000,B 90.000,C 0.000} C_DIS
LIN {X 58.131,Y -35.719,Z -40.220,A -90.000,B 90.000,C 0.000} C_DIS
LIN {X 56.731,Y -35.719,Z -39.462,A -90.000,B 90.000,C 0.000} C_DIS
LIN {X 55.623,Y -35.719,Z -38.990,A -90.000,B 90.000,C 0.000} C_DIS
LIN {X 54.497,Y -35.719,Z -38.563,A -90.000,B 90.000,C 0.000} C_DIS
LIN {X 53.354,Y -35.719,Z -38.182,A -90.000,B 90.000,C 0.000} C_DIS
LIN {X 52.196,Y -35.719,Z -37.848,A -90.000,B 90.000,C 0.000} C_DIS
LIN {X 51.027,Y -35.719,Z -37.561,A -90.000,B 90.000,C 0.000} C_DIS
LIN {X 49.846,Y -35.719,Z -37.322,A -90.000,B 90.000,C 0.000} C_DIS
LIN {X 48.570,Y -35.719,Z -37.275,A -90.000,B 90.000,C 0.000} C_DIS
LIN {X 47.293,Y -35.719,Z -37.290,A -90.000,B 90.000,C 0.000} C_DIS
LIN {X 46.018,Y -35.719,Z -37.369,A -90.000,B 90.000,C 0.000} C_DIS
LIN {X 44.749,Y -35.719,Z -37.510,A -90.000,B 90.000,C 0.000} C_DIS
LIN {X 43.488,Y -35.719,Z -37.713,A -90.000,B 90.000,C 0.000} C_DIS
LIN {X 42.239,Y -35.719,Z -37.978,A -90.000,B 90.000,C 0.000} C_DIS
LIN {X 41.004,Y -35.719,Z -38.305,A -90.000,B 90.000,C 0.000} C_DIS
LIN {X 39.219,Y -35.719,Z -38.105,A -90.000,B 90.000,C 0.000} C_DIS
LIN {X 37.430,Y -35.719,Z -37.937,A -90.000,B 90.000,C 0.000} C_DIS
LIN {X 35.639,Y -35.719,Z -37.802,A -90.000,B 90.000,C 0.000} C_DIS
LIN {X 34.523,Y -35.719,Z -37.894,A -90.000,B 90.000,C 0.000} C_DIS
LIN {X 33.416,Y -35.719,Z -38.058,A -90.000,B 90.000,C 0.000} C_DIS
LIN {X 32.321,Y -35.719,Z -38.292,A -90.000,B 90.000,C 0.000} C_DIS
LIN {X 31.244,Y -35.719,Z -38.595,A -90.000,B 90.000,C 0.000} C_DIS
LIN {X 30.188,Y -35.719,Z -38.967,A -90.000,B 90.000,C 0.000} C_DIS
LIN {X 29.158,Y -35.719,Z -39.406,A -90.000,B 90.000,C 0.000} C_DIS
LIN {X 28.158,Y -35.719,Z -39.909,A -90.000,B 90.000,C 0.000} C_DIS
LIN {X 27.193,Y -35.719,Z -40.476,A -90.000,B 90.000,C 0.000} C_DIS
LIN {X 26.266,Y -35.719,Z -41.103,A -90.000,B 90.000,C 0.000} C_DIS
LIN {X 25.381,Y -35.719,Z -41.789,A -90.000,B 90.000,C 0.000} C_DIS
LIN {X 24.733,Y -35.719,Z -42.391,A -90.000,B 90.000,C 0.000} C_DIS
LIN {X 24.123,Y -35.719,Z -43.032,A -90.000,B 90.000,C 0.000} C_DIS
LIN {X 23.556,Y -35.719,Z -43.710,A -90.000,B 90.000,C 0.000} C_DIS
LIN {X 23.032,Y -35.719,Z -44.423,A -90.000,B 90.000,C 0.000} C_DIS
LIN {X 22.554,Y -35.719,Z -45.167,A -90.000,B 90.000,C 0.000} C_DIS
LIN {X 22.124,Y -35.719,Z -45.940,A -90.000,B 90.000,C 0.000} C_DIS
LIN {X 21.743,Y -35.719,Z -46.738,A -90.000,B 90.000,C 0.000} C_DIS
LIN {X 21.413,Y -35.719,Z -47.559,A -90.000,B 90.000,C 0.000} C_DIS
LIN {X 20.793,Y -35.719,Z -48.141,A -90.000,B 90.000,C 0.000} C_DIS
LIN {X 20.219,Y -35.719,Z -48.767,A -90.000,B 90.000,C 0.000} C_DIS
LIN {X 19.693,Y -35.719,Z -49.434,A -90.000,B 90.000,C 0.000} C_DIS
LIN {X 19.217,Y -35.719,Z -50.139,A -90.000,B 90.000,C 0.000} C_DIS
LIN {X 18.796,Y -35.719,Z -50.877,A -90.000,B 90.000,C 0.000} C_DIS
LIN {X 18.721,Y -35.719,Z -51.016,A -90.000,B 90.000,C 0.000} C_DIS
LIN {X 18.481,Y -35.719,Z -51.539,A -90.000,B 90.000,C 0.000} C_DIS
LIN {X 17.922,Y -35.719,Z -51.645,A -90.000,B 90.000,C 0.000} C_DIS
LIN {X 17.370,Y -35.719,Z -51.787,A -90.000,B 90.000,C 0.000} C_DIS
LIN {X 16.829,Y -35.719,Z -51.964,A -90.000,B 90.000,C 0.000} C_DIS
LIN {X 16.301,Y -35.719,Z -52.176,A -90.000,B 90.000,C 0.000} C_DIS
LIN {X 15.455,Y -35.719,Z -52.168,A -90.000,B 90.000,C 0.000} C_DIS
LIN {X 14.611,Y -35.719,Z -52.221,A -90.000,B 90.000,C 0.000} C_DIS
LIN {X 13.772,Y -35.719,Z -52.332,A -90.000,B 90.000,C 0.000} C_DIS
LIN {X 12.943,Y -35.719,Z -52.502,A -90.000,B 90.000,C 0.000} C_DIS
LIN {X 12.129,Y -35.719,Z -52.731,A -90.000,B 90.000,C 0.000} C_DIS
LIN {X 12.039,Y -35.719,Z -52.762,A -90.000,B 90.000,C 0.000} C_DIS
LIN {X 11.322,Y -35.719,Z -52.964,A -90.000,B 90.000,C 0.000} C_DIS
LIN {X 10.620,Y -35.719,Z -53.212,A -90.000,B 90.000,C 0.000} C_DIS
LIN {X 9.935,Y -35.719,Z -53.505,A -90.000,B 90.000,C 0.000} C_DIS
LIN {X 9.271,Y -35.719,Z -53.842,A -90.000,B 90.000,C 0.000} C_DIS
LIN {X 4.444,Y -35.719,Z -53.842,A -90.000,B 90.000,C 0.000} C_DIS
LIN {X 2.542,Y -35.719,Z -54.591,A -90.000,B 90.000,C 0.000} C_DIS
LIN {X 3.866,Y -35.719,Z -54.781,A -90.000,B 90.000,C 0.000} C_DIS
LIN {X 5.197,Y -35.719,Z -54.921,A -90.000,B 90.000,C 0.000} C_DIS
LIN {X 6.532,Y -35.719,Z -55.010,A -90.000,B 90.000,C 0.000} C_DIS
LIN {X 7.869,Y -35.719,Z -55.050,A -90.000,B 90.000,C 0.000} C_DIS
LIN {X 9.207,Y -35.719,Z -55.039,A -90.000,B 90.000,C 0.000} C_DIS
LIN {X 9.793,Y -35.719,Z -54.696,A -90.000,B 90.000,C 0.000} C_DIS
LIN {X 10.399,Y -35.719,Z -54.392,A -90.000,B 90.000,C 0.000} C_DIS
LIN {X 11.024,Y -35.719,Z -54.128,A -90.000,B 90.000,C 0.000} C_DIS
LIN {X 11.665,Y -35.719,Z -53.904,A -90.000,B 90.000,C 0.000} C_DIS
LIN {X 12.319,Y -35.719,Z -53.723,A -90.000,B 90.000,C 0.000} C_DIS
LIN {X 12.442,Y -35.719,Z -53.681,A -90.000,B 90.000,C 0.000} C_DIS
LIN {X 13.233,Y -35.719,Z -53.462,A -90.000,B 90.000,C 0.000} C_DIS
LIN {X 14.038,Y -35.719,Z -53.302,A -90.000,B 90.000,C 0.000} C_DIS
LIN {X 14.852,Y -35.719,Z -53.203,A -90.000,B 90.000,C 0.000} C_DIS
LIN {X 15.672,Y -35.719,Z -53.165,A -90.000,B 90.000,C 0.000} C_DIS
LIN {X 16.492,Y -35.719,Z -53.188,A -90.000,B 90.000,C 0.000} C_DIS
LIN {X 17.002,Y -35.719,Z -52.968,A -90.000,B 90.000,C 0.000} C_DIS
LIN {X 17.526,Y -35.719,Z -52.784,A -90.000,B 90.000,C 0.000} C_DIS
LIN {X 18.062,Y -35.719,Z -52.639,A -90.000,B 90.000,C 0.000} C_DIS
LIN {X 18.607,Y -35.719,Z -52.532,A -90.000,B 90.000,C 0.000} C_DIS
LIN {X 19.158,Y -35.719,Z -52.464,A -90.000,B 90.000,C 0.000} C_DIS
LIN {X 19.616,Y -35.719,Z -51.463,A -90.000,B 90.000,C 0.000} C_DIS
LIN {X 19.679,Y -35.719,Z -51.348,A -90.000,B 90.000,C 0.000} C_DIS
LIN {X 20.018,Y -35.719,Z -50.747,A -90.000,B 90.000,C 0.000} C_DIS
LIN {X 20.397,Y -35.719,Z -50.169,A -90.000,B 90.000,C 0.000} C_DIS
LIN {X 20.813,Y -35.719,Z -49.618,A -90.000,B 90.000,C 0.000} C_DIS
LIN {X 21.264,Y -35.719,Z -49.096,A -90.000,B 90.000,C 0.000} C_DIS
LIN {X 21.750,Y -35.719,Z -48.605,A -90.000,B 90.000,C 0.000} C_DIS
LIN {X 22.266,Y -35.719,Z -48.147,A -90.000,B 90.000,C 0.000} C_DIS
LIN {X 22.569,Y -35.719,Z -47.350,A -90.000,B 90.000,C 0.000} C_DIS
LIN {X 22.923,Y -35.719,Z -46.575,A -90.000,B 90.000,C 0.000} C_DIS
LIN {X 23.327,Y -35.719,Z -45.824,A -90.000,B 90.000,C 0.000} C_DIS
LIN {X 23.779,Y -35.719,Z -45.102,A -90.000,B 90.000,C 0.000} C_DIS
LIN {X 24.278,Y -35.719,Z -44.410,A -90.000,B 90.000,C 0.000} C_DIS
LIN {X 24.820,Y -35.719,Z -43.753,A -90.000,B 90.000,C 0.000} C_DIS
LIN {X 25.405,Y -35.719,Z -43.132,A -90.000,B 90.000,C 0.000} C_DIS
LIN {X 26.028,Y -35.719,Z -42.551,A -90.000,B 90.000,C 0.000} C_DIS
LIN {X 26.857,Y -35.719,Z -41.910,A -90.000,B 90.000,C 0.000} C_DIS
LIN {X 27.726,Y -35.719,Z -41.322,A -90.000,B 90.000,C 0.000} C_DIS
LIN {X 28.630,Y -35.719,Z -40.791,A -90.000,B 90.000,C 0.000} C_DIS
LIN {X 29.566,Y -35.719,Z -40.319,A -90.000,B 90.000,C 0.000} C_DIS
LIN {X 30.530,Y -35.719,Z -39.907,A -90.000,B 90.000,C 0.000} C_DIS
LIN {X 31.518,Y -35.719,Z -39.557,A -90.000,B 90.000,C 0.000} C_DIS
LIN {X 32.526,Y -35.719,Z -39.271,A -90.000,B 90.000,C 0.000} C_DIS
LIN {X 33.551,Y -35.719,Z -39.050,A -90.000,B 90.000,C 0.000} C_DIS
LIN {X 34.588,Y -35.719,Z -38.894,A -90.000,B 90.000,C 0.000} C_DIS
LIN {X 35.632,Y -35.719,Z -38.803,A -90.000,B 90.000,C 0.000} C_DIS
LIN {X 37.454,Y -35.719,Z -38.942,A -90.000,B 90.000,C 0.000} C_DIS
LIN {X 39.273,Y -35.719,Z -39.115,A -90.000,B 90.000,C 0.000} C_DIS
LIN {X 41.089,Y -35.719,Z -39.323,A -90.000,B 90.000,C 0.000} C_DIS
LIN {X 42.293,Y -35.719,Z -38.995,A -90.000,B 90.000,C 0.000} C_DIS
LIN {X 43.513,Y -35.719,Z -38.727,A -90.000,B 90.000,C 0.000} C_DIS
LIN {X 44.744,Y -35.719,Z -38.520,A -90.000,B 90.000,C 0.000} C_DIS
LIN {X 45.984,Y -35.719,Z -38.376,A -90.000,B 90.000,C 0.000} C_DIS
LIN {X 47.230,Y -35.719,Z -38.294,A -90.000,B 90.000,C 0.000} C_DIS
LIN {X 48.478,Y -35.719,Z -38.274,A -90.000,B 90.000,C 0.000} C_DIS
LIN {X 49.726,Y -35.719,Z -38.317,A -90.000,B 90.000,C 0.000} C_DIS
LIN {X 50.852,Y -35.719,Z -38.547,A -90.000,B 90.000,C 0.000} C_DIS
LIN {X 51.969,Y -35.719,Z -38.823,A -90.000,B 90.000,C 0.000} C_DIS
LIN {X 53.073,Y -35.719,Z -39.142,A -90.000,B 90.000,C 0.000} C_DIS
LIN {X 54.164,Y -35.719,Z -39.506,A -90.000,B 90.000,C 0.000} C_DIS
LIN {X 55.239,Y -35.719,Z -39.913,A -90.000,B 90.000,C 0.000} C_DIS
LIN {X 56.297,Y -35.719,Z -40.363,A -90.000,B 90.000,C 0.000} C_DIS
LIN {X 57.655,Y -35.719,Z -41.100,A -90.000,B 90.000,C 0.000} C_DIS
LIN {X 58.979,Y -35.719,Z -41.895,A -90.000,B 90.000,C 0.000} C_DIS
LIN {X 60.268,Y -35.719,Z -42.746,A -90.000,B 90.000,C 0.000} C_DIS
LIN {X 61.518,Y -35.719,Z -43.653,A -90.000,B 90.000,C 0.000} C_DIS
LIN {X 62.728,Y -35.719,Z -44.613,A -90.000,B 90.000,C 0.000} C_DIS
LIN {X 63.895,Y -35.719,Z -45.624,A -90.000,B 90.000,C 0.000} C_DIS
LIN {X 65.017,Y -35.719,Z -46.686,A -90.000,B 90.000,C 0.000} C_DIS
LIN {X 66.531,Y -35.719,Z -48.146,A -90.000,B 90.000,C 0.000} C_DIS
LIN {X 68.071,Y -35.719,Z -49.578,A -90.000,B 90.000,C 0.000} C_DIS
LIN {X 69.637,Y -35.719,Z -50.981,A -90.000,B 90.000,C 0.000} C_DIS
LIN {X 71.229,Y -35.719,Z -52.356,A -90.000,B 90.000,C 0.000} C_DIS
LIN {X 72.289,Y -35.719,Z -53.216,A -90.000,B 90.000,C 0.000} C_DIS
LIN {X 73.314,Y -35.719,Z -54.119,A -90.000,B 90.000,C 0.000} C_DIS
LIN {X 74.301,Y -35.719,Z -55.061,A -90.000,B 90.000,C 0.000} C_DIS
LIN {X 75.250,Y -35.719,Z -56.043,A -90.000,B 90.000,C 0.000} C_DIS
LIN {X 76.159,Y -35.719,Z -57.062,A -90.000,B 90.000,C 0.000} C_DIS
LIN {X 77.026,Y -35.719,Z -58.116,A -90.000,B 90.000,C 0.000} C_DIS
LIN {X 78.176,Y -35.719,Z -56.565,A -90.000,B 90.000,C 0.000} C_DIS
LIN {X 79.375,Y -35.719,Z -55.053,A -90.000,B 90.000,C 0.000} C_DIS
LIN {X 80.624,Y -35.719,Z -53.581,A -90.000,B 90.000,C 0.000} C_DIS
LIN {X 81.920,Y -35.719,Z -52.150,A -90.000,B 90.000,C 0.000} C_DIS
LIN {X 83.263,Y -35.719,Z -50.763,A -90.000,B 90.000,C 0.000} C_DIS
LIN {X 84.650,Y -35.719,Z -49.421,A -90.000,B 90.000,C 0.000} C_DIS
LIN {X 86.081,Y -35.719,Z -48.125,A -90.000,B 90.000,C 0.000} C_DIS
LIN {X 86.021,Y -35.719,Z -47.509,A -90.000,B 90.000,C 0.000} C_DIS
LIN {X 86.001,Y -35.719,Z -46.891,A -90.000,B 90.000,C 0.000} C_DIS
LIN {X 86.021,Y -35.719,Z -46.273,A -90.000,B 90.000,C 0.000} C_DIS
LIN {X 86.081,Y -35.719,Z -45.657,A -90.000,B 90.000,C 0.000} C_DIS
LIN {X 86.180,Y -35.719,Z -45.047,A -90.000,B 90.000,C 0.000} C_DIS
LIN {X 86.438,Y -35.719,Z -44.026,A -90.000,B 90.000,C 0.000} C_DIS
LIN {X 86.762,Y -35.719,Z -43.024,A -90.000,B 90.000,C 0.000} C_DIS
LIN {X 87.152,Y -35.719,Z -42.045,A -90.000,B 90.000,C 0.000} C_DIS
LIN {X 87.605,Y -35.719,Z -41.095,A -90.000,B 90.000,C 0.000} C_DIS
LIN {X 88.120,Y -35.719,Z -40.176,A -90.000,B 90.000,C 0.000} C_DIS
LIN {X 88.694,Y -35.719,Z -39.293,A -90.000,B 90.000,C 0.000} C_DIS
LIN {X 89.326,Y -35.719,Z -38.450,A -90.000,B 90.000,C 0.000} C_DIS
LIN {X 90.011,Y -35.719,Z -37.651,A -90.000,B 90.000,C 0.000} C_DIS
LIN {X 90.748,Y -35.719,Z -36.898,A -90.000,B 90.000,C 0.000} C_DIS
LIN {X 91.532,Y -35.719,Z -36.195,A -90.000,B 90.000,C 0.000} C_DIS
LIN {X 92.362,Y -35.719,Z -35.546,A -90.000,B 90.000,C 0.000} C_DIS
LIN {X 93.232,Y -35.719,Z -34.953,A -90.000,B 90.000,C 0.000} C_DIS
LIN {X 95.062,Y -35.719,Z -33.941,A -90.000,B 90.000,C 0.000} C_DIS
LIN {X 96.918,Y -35.719,Z -32.978,A -90.000,B 90.000,C 0.000} C_DIS
LIN {X 98.798,Y -35.719,Z -32.063,A -90.000,B 90.000,C 0.000} C_DIS
LIN {X 100.701,Y -35.719,Z -31.198,A -90.000,B 90.000,C 0.000} C_DIS
LIN {X 102.627,Y -35.719,Z -30.382,A -90.000,B 90.000,C 0.000} C_DIS
LIN {X 104.573,Y -35.719,Z -29.618,A -90.000,B 90.000,C 0.000} C_DIS
LIN {X 105.509,Y -35.719,Z -29.233,A -90.000,B 90.000,C 0.000} C_DIS
LIN {X 106.470,Y -35.719,Z -28.914,A -90.000,B 90.000,C 0.000} C_DIS
LIN {X 107.452,Y -35.719,Z -28.665,A -90.000,B 90.000,C 0.000} C_DIS
LIN {X 108.448,Y -35.719,Z -28.486,A -90.000,B 90.000,C 0.000} C_DIS
LIN {X 109.455,Y -35.719,Z -28.377,A -90.000,B 90.000,C 0.000} C_DIS
LIN {X 110.466,Y -35.719,Z -28.340,A -90.000,B 90.000,C 0.000} C_DIS
LIN {X 111.478,Y -35.719,Z -28.375,A -90.000,B 90.000,C 0.000} C_DIS
LIN {X 112.485,Y -35.719,Z -28.481,A -90.000,B 90.000,C 0.000} C_DIS
LIN {X 113.482,Y -35.719,Z -28.658,A -90.000,B 90.000,C 0.000} C_DIS
LIN {X 114.464,Y -35.719,Z -28.906,A -90.000,B 90.000,C 0.000} C_DIS
LIN {X 115.426,Y -35.719,Z -29.222,A -90.000,B 90.000,C 0.000} C_DIS
LIN {X 116.363,Y -35.719,Z -29.605,A -90.000,B 90.000,C 0.000} C_DIS
LIN {X 117.270,Y -35.719,Z -30.054,A -90.000,B 90.000,C 0.000} C_DIS
LIN {X 118.144,Y -35.719,Z -30.566,A -90.000,B 90.000,C 0.000} C_DIS
LIN {X 118.979,Y -35.719,Z -31.138,A -90.000,B 90.000,C 0.000} C_DIS
LIN {X 119.134,Y -35.719,Z -31.254,A -90.000,B 90.000,C 0.000} C_DIS
LIN {X 119.802,Y -35.719,Z -31.812,A -90.000,B 90.000,C 0.000} C_DIS
LIN {X 120.437,Y -35.719,Z -32.407,A -90.000,B 90.000,C 0.000} C_DIS
LIN {X 121.037,Y -35.719,Z -33.038,A -90.000,B 90.000,C 0.000} C_DIS
LIN {X 121.600,Y -35.719,Z -33.701,A -90.000,B 90.000,C 0.000} C_DIS
LIN {X 121.662,Y -35.719,Z -33.780,A -90.000,B 90.000,C 0.000} C_DIS
LIN {X 122.196,Y -35.719,Z -34.612,A -90.000,B 90.000,C 0.000} C_DIS
LIN {X 122.676,Y -35.719,Z -35.476,A -90.000,B 90.000,C 0.000} C_DIS
LIN {X 123.102,Y -35.719,Z -36.368,A -90.000,B 90.000,C 0.000} C_DIS
LIN {X 123.470,Y -35.719,Z -37.286,A -90.000,B 90.000,C 0.000} C_DIS
LIN {X 123.781,Y -35.719,Z -38.224,A -90.000,B 90.000,C 0.000} C_DIS
LIN {X 124.032,Y -35.719,Z -39.180,A -90.000,B 90.000,C 0.000} C_DIS
LIN {X 124.222,Y -35.719,Z -40.150,A -90.000,B 90.000,C 0.000} C_DIS
LIN {X 124.352,Y -35.719,Z -41.130,A -90.000,B 90.000,C 0.000} C_DIS
LIN {X 124.419,Y -35.719,Z -42.117,A -90.000,B 90.000,C 0.000} C_DIS
LIN {X 124.425,Y -35.719,Z -43.105,A -90.000,B 90.000,C 0.000} C_DIS
LIN {X 124.369,Y -35.719,Z -44.092,A -90.000,B 90.000,C 0.000} C_DIS
LIN {X 124.170,Y -35.719,Z -45.366,A -90.000,B 90.000,C 0.000} C_DIS
LIN {X 123.911,Y -35.719,Z -46.630,A -90.000,B 90.000,C 0.000} C_DIS
LIN {X 123.595,Y -35.719,Z -47.880,A -90.000,B 90.000,C 0.000} C_DIS
LIN {X 123.220,Y -35.719,Z -49.114,A -90.000,B 90.000,C 0.000} C_DIS
LIN {X 122.789,Y -35.719,Z -50.330,A -90.000,B 90.000,C 0.000} C_DIS
LIN {X 122.302,Y -35.719,Z -51.524,A -90.000,B 90.000,C 0.000} C_DIS
LIN {X 121.760,Y -35.719,Z -52.694,A -90.000,B 90.000,C 0.000} C_DIS
LIN {X 121.019,Y -35.719,Z -54.060,A -90.000,B 90.000,C 0.000} C_DIS
LIN {X 120.326,Y -35.719,Z -55.451,A -90.000,B 90.000,C 0.000} C_DIS
LIN {X 119.682,Y -35.719,Z -56.866,A -90.000,B 90.000,C 0.000} C_DIS
LIN {X 119.089,Y -35.719,Z -58.302,A -90.000,B 90.000,C 0.000} C_DIS
LIN {X 118.546,Y -35.719,Z -59.759,A -90.000,B 90.000,C 0.000} C_DIS
LIN {X 118.055,Y -35.719,Z -61.233,A -90.000,B 90.000,C 0.000} C_DIS
LIN {X 117.477,Y -35.719,Z -63.546,A -90.000,B 90.000,C 0.000} C_DIS
